LIN {X 0,Y 262.257,Z 673.457,A -85,B 0,C 180,E1 -18836.778,E2 -18836.778} C_VEL
LIN {X 0,Y 264.045,Z 616.117,A -85,B 0,C 180,E1 -18838.311,E2 -18838.311} C_VEL
LIN {X 0,Y 260.574,Z 590.625,A -85,B 0,C 180,E1 -18839.463,E2 -18839.463} C_VEL
LIN {X 0,Y 259.509,Z 585.684,A -85,B 0,C 180,E1 -18839.736,E2 -18839.736} C_VEL
LIN {X 0,Y 253.189,Z 570.092,A -85,B 0,C 180,E1 -18840.985,E2 -18840.985} C_VEL
LIN {X 0,Y 252.204,Z 567.395,A -85,B 0,C 180,E1 -18841.255,E2 -18841.255} C_VEL
LIN {X 0,Y 250.326,Z 558.805,A -85,B 0,C 180,E1 -18844.748,E2 -18844.748} C_VEL
LIN {X 0,Y 249.114,Z 553.456,A -85,B 0,C 180,E1 -18847.086,E2 -18847.086} C_VEL
LIN {X 0,Y 249.024,Z 553.465,A -85,B 0,C 180,E1 -18850.473,E2 -18850.473} C_VEL
LIN {X 0,Y 249.007,Z 553.466,A -85,B 0,C 180,E1 -18854.877,E2 -18854.877} C_VEL
LIN {X 0,Y 249.027,Z 553.464,A -85,B 0,C 180,E1 -18857.365,E2 -18857.365} C_VEL
LIN {X 0,Y 249.047,Z 553.463,A -85,B 0,C 180,E1 -18861.623,E2 -18861.623} C_VEL
LIN {X 0,Y 249.057,Z 553.461,A -85,B 0,C 180,E1 -18865.642,E2 -18865.642} C_VEL
LIN {X 0,Y 249.048,Z 553.464,A -85,B 0,C 180,E1 -18869.473,E2 -18869.473} C_VEL
LIN {X 0,Y 249.065,Z 553.457,A -85,B 0,C 180,E1 -18873.161,E2 -18873.161} C_VEL
LIN {X 0,Y 249.056,Z 553.455,A -85,B 0,C 180,E1 -18876.73,E2 -18876.73} C_VEL
LIN {X 0,Y 249.102,Z 553.454,A -85,B 0,C 180,E1 -18880.211,E2 -18880.211} C_VEL
LIN {X 0,Y 249.218,Z 553.438,A -85,B 0,C 180,E1 -18883.62,E2 -18883.62} C_VEL
LIN {X 0,Y 249.247,Z 553.429,A -85,B 0,C 180,E1 -18888.616,E2 -18888.616} C_VEL
LIN {X 0,Y 249.474,Z 553.409,A -85,B 0,C 180,E1 -18891.903,E2 -18891.903} C_VEL
LIN {X 0,Y 249.43,Z 553.409,A -85,B 0,C 180,E1 -18896.77,E2 -18896.77} C_VEL
LIN {X 0,Y 249.722,Z 553.376,A -85,B 0,C 180,E1 -18900,E2 -18900} C_VEL
LIN {X 0,Y 249.43,Z 553.406,A -85,B 0,C 180,E1 -18903.231,E2 -18903.231} C_VEL
LIN {X 0,Y 249.436,Z 553.41,A -85,B 0,C 180,E1 -18906.71,E2 -18906.71} C_VEL
LIN {X 0,Y 249.338,Z 553.412,A -85,B 0,C 180,E1 -18909.737,E2 -18909.737} C_VEL
LIN {X 0,Y 249.196,Z 553.442,A -85,B 0,C 180,E1 -18914.704,E2 -18914.704} C_VEL
LIN {X 0,Y 249.134,Z 553.444,A -85,B 0,C 180,E1 -18918.078,E2 -18918.078} C_VEL
LIN {X 0,Y 249.084,Z 553.449,A -85,B 0,C 180,E1 -18921.519,E2 -18921.519} C_VEL
LIN {X 0,Y 249.127,Z 553.451,A -85,B 0,C 180,E1 -18925.483,E2 -18925.483} C_VEL
LIN {X 0,Y 249.08,Z 553.458,A -85,B 0,C 180,E1 -18928.994,E2 -18928.994} C_VEL
LIN {X 0,Y 249.033,Z 553.461,A -85,B 0,C 180,E1 -18932.426,E2 -18932.426} C_VEL
LIN {X 0,Y 249.065,Z 553.451,A -85,B 0,C 180,E1 -18936.34,E2 -18936.34} C_VEL
LIN {X 0,Y 249.026,Z 553.463,A -85,B 0,C 180,E1 -18940.475,E2 -18940.475} C_VEL
LIN {X 0,Y 249.018,Z 553.466,A -85,B 0,C 180,E1 -18944.876,E2 -18944.876} C_VEL
LIN {X 0,Y 249.061,Z 553.462,A -85,B 0,C 180,E1 -18947.374,E2 -18947.374} C_VEL
LIN {X 0,Y 249.053,Z 553.46,A -85,B 0,C 180,E1 -18951.625,E2 -18951.625} C_VEL
LIN {X 0,Y 249.062,Z 553.46,A -85,B 0,C 180,E1 -18955.643,E2 -18955.643} C_VEL
LIN {X 0,Y 249.053,Z 553.464,A -85,B 0,C 180,E1 -18959.474,E2 -18959.474} C_VEL
LIN {X 0,Y 249.126,Z 553.516,A -85,B 0,C 180,E1 -18961.618,E2 -18961.618} C_VEL
LIN {X 0,Y 249.669,Z 555.641,A -85,B 0,C 180,E1 -18962.555,E2 -18962.555} C_VEL
LIN {X 0,Y 258.002,Z 574.299,A -85,B 0,C 180,E1 -18964.192,E2 -18964.192} C_VEL
LIN {X 0,Y 264.581,Z 591.655,A -85,B 0,C 180,E1 -18965.475,E2 -18965.475} C_VEL
LIN {X 0,Y 264.668,Z 597.246,A -85,B 0,C 180,E1 -18965.651,E2 -18965.651} C_VEL
LIN {X 0,Y 262.519,Z 662.1,A -85,B 0,C 180,E1 -18967.389,E2 -18967.389} C_VEL
LIN {X 0,Y 261.67,Z 674.994,A -85,B 0,C 180,E1 -18968.017,E2 -18968.017} C_VEL
LIN {X 0,Y 260.478,Z 687.741,A -85,B 0,C 180,E1 -18968.95,E2 -18968.95} C_VEL
LIN {X 0,Y 258.823,Z 699.889,A -85,B 0,C 180,E1 -18970.159,E2 -18970.159} C_VEL
LIN {X 0,Y 257.099,Z 711.369,A -85,B 0,C 180,E1 -18971.678,E2 -18971.678} C_VEL
LIN {X 0,Y 255.207,Z 721.715,A -85,B 0,C 180,E1 -18973.399,E2 -18973.399} C_VEL
LIN {X 0,Y 253.426,Z 730.182,A -85,B 0,C 180,E1 -18975.137,E2 -18975.137} C_VEL
LIN {X 0,Y 251.969,Z 737.973,A -85,B 0,C 180,E1 -18977.107,E2 -18977.107} C_VEL
LIN {X 0,Y 250.533,Z 745.289,A -85,B 0,C 180,E1 -18979.383,E2 -18979.383} C_VEL
LIN {X 0,Y 249.222,Z 751.71,A -85,B 0,C 180,E1 -18981.895,E2 -18981.895} C_VEL
LIN {X 0,Y 248.21,Z 756.578,A -85,B 0,C 180,E1 -18984.313,E2 -18984.313} C_VEL
LIN {X 0,Y 247.435,Z 760.339,A -85,B 0,C 180,E1 -18986.744,E2 -18986.744} C_VEL
LIN {X 0,Y 247.176,Z 762.276,A -85,B 0,C 180,E1 -18988.371,E2 -18988.371} C_VEL
LIN {X 0,Y 247.031,Z 763.804,A -85,B 0,C 180,E1 -18990,E2 -18990} C_VEL
LIN {X 0,Y 246.982,Z 764.891,A -85,B 0,C 180,E1 -18991.631,E2 -18991.631} C_VEL
LIN {X 0,Y 246.929,Z 765.58,A -85,B 0,C 180,E1 -18993.263,E2 -18993.263} C_VEL
LIN {X 0,Y 246.946,Z 765.908,A -85,B 0,C 180,E1 -18995.063,E2 -18995.063} C_VEL
LIN {X 0,Y 247.097,Z 765.335,A -85,B 0,C 180,E1 -18998.176,E2 -18998.176} C_VEL
LIN {X 0,Y 247.641,Z 763.152,A -85,B 0,C 180,E1 -19001.458,E2 -19001.458} C_VEL
LIN {X 0,Y 248.453,Z 760.413,A -85,B 0,C 180,E1 -19003.912,E2 -19003.912} C_VEL
LIN {X 0,Y 249.557,Z 756.648,A -85,B 0,C 180,E1 -19006.356,E2 -19006.356} C_VEL
LIN {X 0,Y 250.927,Z 751.748,A -85,B 0,C 180,E1 -19008.789,E2 -19008.789} C_VEL
LIN {X 0,Y 252.776,Z 745.563,A -85,B 0,C 180,E1 -19011.188,E2 -19011.188} C_VEL
LIN {X 0,Y 255.064,Z 737.823,A -85,B 0,C 180,E1 -19013.548,E2 -19013.548} C_VEL
LIN {X 0,Y 257.084,Z 729.651,A -85,B 0,C 180,E1 -19015.559,E2 -19015.559} C_VEL
LIN {X 0,Y 259.657,Z 719.105,A -85,B 0,C 180,E1 -19017.613,E2 -19017.613} C_VEL
LIN {X 0,Y 262.078,Z 707.972,A -85,B 0,C 180,E1 -19019.3,E2 -19019.3} C_VEL
LIN {X 0,Y 264.16,Z 697.037,A -85,B 0,C 180,E1 -19020.585,E2 -19020.585} C_VEL
LIN {X 0,Y 265.809,Z 684.913,A -85,B 0,C 180,E1 -19021.701,E2 -19021.701} C_VEL
LIN {X 0,Y 267.279,Z 672.232,A -85,B 0,C 180,E1 -19022.515,E2 -19022.515} C_VEL
LIN {X 0,Y 268.122,Z 659.678,A -85,B 0,C 180,E1 -19023.043,E2 -19023.043} C_VEL
LIN {X 0,Y 270.333,Z 598.373,A -85,B 0,C 180,E1 -19024.656,E2 -19024.656} C_VEL
LIN {X 0,Y 262.528,Z 580.576,A -85,B 0,C 180,E1 -19026.328,E2 -19026.328} C_VEL
LIN {X 0,Y 255.474,Z 566.537,A -85,B 0,C 180,E1 -19027.89,E2 -19027.89} C_VEL
LIN {X 0,Y 251.234,Z 559.018,A -85,B 0,C 180,E1 -19028.855,E2 -19028.855} C_VEL
LIN {X 0,Y 249.654,Z 555.862,A -85,B 0,C 180,E1 -19029.271,E2 -19029.271} C_VEL
LIN {X 0,Y 249.064,Z 553.462,A -85,B 0,C 180,E1 -19030.598,E2 -19030.598} C_VEL
LIN {X 0,Y 249.021,Z 553.465,A -85,B 0,C 180,E1 -19034.874,E2 -19034.874} C_VEL
LIN {X 0,Y 249.052,Z 553.456,A -85,B 0,C 180,E1 -19037.37,E2 -19037.37} C_VEL
LIN {X 0,Y 249.063,Z 553.46,A -85,B 0,C 180,E1 -19042.193,E2 -19042.193} C_VEL
LIN {X 0,Y 249.059,Z 553.457,A -85,B 0,C 180,E1 -19045.641,E2 -19045.641} C_VEL
LIN {X 0,Y 249.049,Z 553.454,A -85,B 0,C 180,E1 -19049.472,E2 -19049.472} C_VEL
LIN {X 0,Y 249.07,Z 553.451,A -85,B 0,C 180,E1 -19053.161,E2 -19053.161} C_VEL
LIN {X 0,Y 249.075,Z 553.453,A -85,B 0,C 180,E1 -19056.732,E2 -19056.732} C_VEL
LIN {X 0,Y 249.106,Z 553.456,A -85,B 0,C 180,E1 -19060.211,E2 -19060.211} C_VEL
LIN {X 0,Y 249.238,Z 553.436,A -85,B 0,C 180,E1 -19063.621,E2 -19063.621} C_VEL
LIN {X 0,Y 249.239,Z 553.433,A -85,B 0,C 180,E1 -19068.616,E2 -19068.616} C_VEL
LIN {X 0,Y 249.449,Z 553.402,A -85,B 0,C 180,E1 -19071.902,E2 -19071.902} C_VEL
LIN {X 0,Y 249.293,Z 553.432,A -85,B 0,C 180,E1 -19075.148,E2 -19075.148} C_VEL
LIN {X 0,Y 249.671,Z 553.373,A -85,B 0,C 180,E1 -19078.387,E2 -19078.387} C_VEL
LIN {X 0,Y 249.67,Z 553.382,A -85,B 0,C 180,E1 -19081.613,E2 -19081.613} C_VEL
LIN {X 0,Y 249.423,Z 553.408,A -85,B 0,C 180,E1 -19087.191,E2 -19087.191} C_VEL
LIN {X 0,Y 248.731,Z 553.493,A -85,B 0,C 180,E1 -19088.537,E2 -19088.537} C_VEL
LIN {X 0,Y 245.778,Z 553.87,A -85,B 0,C 180,E1 -19090.729,E2 -19090.729} C_VEL
LIN {X 0,Y 243.276,Z 554.174,A -85,B 0,C 180,E1 -19092.515,E2 -19092.515} C_VEL
LIN {X 0,Y 242.212,Z 554.302,A -85,B 0,C 180,E1 -19093.903,E2 -19093.903} C_VEL
LIN {X 0,Y 242.131,Z 554.314,A -85,B 0,C 180,E1 -19094.374,E2 -19094.374} C_VEL
LIN {X 0,Y 242.146,Z 554.32,A -85,B 0,C 180,E1 -19096.872,E2 -19096.872} C_VEL
LIN {X 0,Y 242.021,Z 554.336,A -85,B 0,C 180,E1 -19101.687,E2 -19101.687} C_VEL
LIN {X 0,Y 242.062,Z 554.332,A -85,B 0,C 180,E1 -19105.838,E2 -19105.838} C_VEL
LIN {X 0,Y 242.026,Z 554.336,A -85,B 0,C 180,E1 -19109.581,E2 -19109.581} C_VEL
LIN {X 0,Y 241.987,Z 554.341,A -85,B 0,C 180,E1 -19113.491,E2 -19113.491} C_VEL
LIN {X 0,Y 242.008,Z 554.339,A -85,B 0,C 180,E1 -19117.578,E2 -19117.578} C_VEL
LIN {X 0,Y 241.953,Z 554.348,A -85,B 0,C 180,E1 -19121.919,E2 -19121.919} C_VEL
LIN {X 0,Y 241.935,Z 554.351,A -85,B 0,C 180,E1 -19126.571,E2 -19126.571} C_VEL
LIN {X 0,Y 241.991,Z 554.486,A -85,B 0,C 180,E1 -19127.942,E2 -19127.942} C_VEL
LIN {X 0,Y 244.207,Z 562.602,A -85,B 0,C 180,E1 -19132.006,E2 -19132.006} C_VEL
LIN {X 0,Y 245.342,Z 567.185,A -85,B 0,C 180,E1 -19134.048,E2 -19134.048} C_VEL
LIN {X 0,Y 254.461,Z 585.606,A -85,B 0,C 180,E1 -19136.239,E2 -19136.239} C_VEL
LIN {X 0,Y 260.641,Z 599.85,A -85,B 0,C 180,E1 -19137.663,E2 -19137.663} C_VEL
LIN {X 0,Y 263.653,Z 619.289,A -85,B 0,C 180,E1 -19138.723,E2 -19138.723} C_VEL
LIN {X 0,Y 261.5,Z 675.447,A -85,B 0,C 180,E1 -19140.247,E2 -19140.247} C_VEL
LIN {X 0,Y 260.259,Z 688.736,A -85,B 0,C 180,E1 -19140.872,E2 -19140.872} C_VEL
LIN {X 0,Y 258.437,Z 701.888,A -85,B 0,C 180,E1 -19141.804,E2 -19141.804} C_VEL
LIN {X 0,Y 256.5,Z 713.038,A -85,B 0,C 180,E1 -19142.902,E2 -19142.902} C_VEL
LIN {X 0,Y 254.106,Z 724.62,A -85,B 0,C 180,E1 -19144.396,E2 -19144.396} C_VEL
LIN {X 0,Y 251.548,Z 735.052,A -85,B 0,C 180,E1 -19146.102,E2 -19146.102} C_VEL
LIN {X 0,Y 249.025,Z 744.458,A -85,B 0,C 180,E1 -19148.042,E2 -19148.042} C_VEL
LIN {X 0,Y 246.902,Z 752.18,A -85,B 0,C 180,E1 -19150.028,E2 -19150.028} C_VEL
LIN {X 0,Y 244.783,Z 759.746,A -85,B 0,C 180,E1 -19152.455,E2 -19152.455} C_VEL
LIN {X 0,Y 242.964,Z 765.844,A -85,B 0,C 180,E1 -19154.91,E2 -19154.91} C_VEL
LIN {X 0,Y 241.589,Z 770.69,A -85,B 0,C 180,E1 -19157.398,E2 -19157.398} C_VEL
LIN {X 0,Y 240.678,Z 774.427,A -85,B 0,C 180,E1 -19159.91,E2 -19159.91} C_VEL
LIN {X 0,Y 240.233,Z 776.363,A -85,B 0,C 180,E1 -19161.589,E2 -19161.589} C_VEL
LIN {X 0,Y 239.956,Z 777.877,A -85,B 0,C 180,E1 -19163.272,E2 -19163.272} C_VEL
LIN {X 0,Y 239.769,Z 779.626,A -85,B 0,C 180,E1 -19166.639,E2 -19166.639} C_VEL
LIN {X 0,Y 239.837,Z 779.923,A -85,B 0,C 180,E1 -19168.321,E2 -19168.321} C_VEL
LIN {X 0,Y 239.915,Z 779.827,A -85,B 0,C 180,E1 -19170,E2 -19170} C_VEL
LIN {X 0,Y 239.841,Z 779.29,A -85,B 0,C 180,E1 -19171.679,E2 -19171.679} C_VEL
LIN {X 0,Y 239.84,Z 777.123,A -85,B 0,C 180,E1 -19174.931,E2 -19174.931} C_VEL
LIN {X 0,Y 240.045,Z 774.202,A -85,B 0,C 180,E1 -19177.571,E2 -19177.571} C_VEL
LIN {X 0,Y 240.553,Z 770.345,A -85,B 0,C 180,E1 -19180.096,E2 -19180.096} C_VEL
LIN {X 0,Y 241.388,Z 765.354,A -85,B 0,C 180,E1 -19182.613,E2 -19182.613} C_VEL
LIN {X 0,Y 242.695,Z 759.08,A -85,B 0,C 180,E1 -19185.107,E2 -19185.107} C_VEL
LIN {X 0,Y 244.409,Z 751.231,A -85,B 0,C 180,E1 -19187.573,E2 -19187.573} C_VEL
LIN {X 0,Y 246.082,Z 742.93,A -85,B 0,C 180,E1 -19189.674,E2 -19189.674} C_VEL
LIN {X 0,Y 247.92,Z 733.413,A -85,B 0,C 180,E1 -19191.624,E2 -19191.624} C_VEL
LIN {X 0,Y 249.979,Z 722.522,A -85,B 0,C 180,E1 -19193.397,E2 -19193.397} C_VEL
LIN {X 0,Y 251.772,Z 711.865,A -85,B 0,C 180,E1 -19194.753,E2 -19194.753} C_VEL
LIN {X 0,Y 253.45,Z 700.16,A -85,B 0,C 180,E1 -19195.895,E2 -19195.895} C_VEL
LIN {X 0,Y 254.928,Z 686.874,A -85,B 0,C 180,E1 -19196.835,E2 -19196.835} C_VEL
LIN {X 0,Y 255.794,Z 674.748,A -85,B 0,C 180,E1 -19197.4,E2 -19197.4} C_VEL
LIN {X 0,Y 257.705,Z 617.043,A -85,B 0,C 180,E1 -19198.982,E2 -19198.982} C_VEL
LIN {X 0,Y 253.937,Z 589.557,A -85,B 0,C 180,E1 -19200.278,E2 -19200.278} C_VEL
LIN {X 0,Y 247.922,Z 574.236,A -85,B 0,C 180,E1 -19201.526,E2 -19201.526} C_VEL
LIN {X 0,Y 244.945,Z 567.249,A -85,B 0,C 180,E1 -19202.186,E2 -19202.186} C_VEL
LIN {X 0,Y 243.05,Z 558.388,A -85,B 0,C 180,E1 -19205.939,E2 -19205.939} C_VEL
LIN {X 0,Y 242.015,Z 554.34,A -85,B 0,C 180,E1 -19207.772,E2 -19207.772} C_VEL
LIN {X 0,Y 241.942,Z 554.346,A -85,B 0,C 180,E1 -19211.92,E2 -19211.92} C_VEL
LIN {X 0,Y 241.942,Z 554.344,A -85,B 0,C 180,E1 -19216.568,E2 -19216.568} C_VEL
LIN {X 0,Y 241.985,Z 554.34,A -85,B 0,C 180,E1 -19220.287,E2 -19220.287} C_VEL
LIN {X 0,Y 242.033,Z 554.334,A -85,B 0,C 180,E1 -19224.497,E2 -19224.497} C_VEL
LIN {X 0,Y 241.972,Z 554.341,A -85,B 0,C 180,E1 -19228.48,E2 -19228.48} C_VEL
LIN {X 0,Y 242.002,Z 554.334,A -85,B 0,C 180,E1 -19232.312,E2 -19232.312} C_VEL
LIN {X 0,Y 242.036,Z 554.33,A -85,B 0,C 180,E1 -19236.014,E2 -19236.014} C_VEL
LIN {X 0,Y 242.03,Z 554.338,A -85,B 0,C 180,E1 -19239.607,E2 -19239.607} C_VEL
LIN {X 0,Y 242.159,Z 554.314,A -85,B 0,C 180,E1 -19243.278,E2 -19243.278} C_VEL
LIN {X 0,Y 242.18,Z 554.309,A -85,B 0,C 180,E1 -19248.28,E2 -19248.28} C_VEL
LIN {X 0,Y 242.421,Z 554.289,A -85,B 0,C 180,E1 -19251.666,E2 -19251.666} C_VEL
LIN {X 0,Y 242.253,Z 554.301,A -85,B 0,C 180,E1 -19255.007,E2 -19255.007} C_VEL
LIN {X 0,Y 242.631,Z 554.26,A -85,B 0,C 180,E1 -19258.34,E2 -19258.34} C_VEL
LIN {X 0,Y 242.631,Z 554.253,A -85,B 0,C 180,E1 -19261.66,E2 -19261.66} C_VEL
LIN {X 0,Y 242.417,Z 554.287,A -85,B 0,C 180,E1 -19266.682,E2 -19266.682} C_VEL
LIN {X 0,Y 242.262,Z 554.291,A -85,B 0,C 180,E1 -19270.024,E2 -19270.024} C_VEL
LIN {X 0,Y 242.159,Z 554.32,A -85,B 0,C 180,E1 -19275.142,E2 -19275.142} C_VEL
LIN {X 0,Y 242.068,Z 554.323,A -85,B 0,C 180,E1 -19278.625,E2 -19278.625} C_VEL
LIN {X 0,Y 242.01,Z 554.335,A -85,B 0,C 180,E1 -19282.181,E2 -19282.181} C_VEL
LIN {X 0,Y 242.063,Z 554.328,A -85,B 0,C 180,E1 -19285.839,E2 -19285.839} C_VEL
LIN {X 0,Y 242.027,Z 554.337,A -85,B 0,C 180,E1 -19289.581,E2 -19289.581} C_VEL
LIN {X 0,Y 241.988,Z 554.344,A -85,B 0,C 180,E1 -19293.492,E2 -19293.492} C_VEL
LIN {X 0,Y 241.996,Z 554.325,A -85,B 0,C 180,E1 -19297.581,E2 -19297.581} C_VEL
LIN {X 0,Y 241.951,Z 554.345,A -85,B 0,C 180,E1 -19301.92,E2 -19301.92} C_VEL
LIN {X 0,Y 241.99,Z 554.338,A -85,B 0,C 180,E1 -19306.558,E2 -19306.558} C_VEL
LIN {X 0,Y 242.008,Z 554.337,A -85,B 0,C 180,E1 -19310.292,E2 -19310.292} C_VEL
LIN {X 0,Y 242.037,Z 554.335,A -85,B 0,C 180,E1 -19314.499,E2 -19314.499} C_VEL
LIN {X 0,Y 241.977,Z 554.345,A -85,B 0,C 180,E1 -19318.481,E2 -19318.481} C_VEL
LIN {X 0,Y 242.044,Z 554.361,A -85,B 0,C 180,E1 -19320.899,E2 -19320.899} C_VEL
LIN {X 0,Y 242.432,Z 555.851,A -85,B 0,C 180,E1 -19321.575,E2 -19321.575} C_VEL
LIN {X 0,Y 250.422,Z 573.112,A -85,B 0,C 180,E1 -19323.218,E2 -19323.218} C_VEL
LIN {X 0,Y 258.393,Z 593.558,A -85,B 0,C 180,E1 -19324.833,E2 -19324.833} C_VEL
LIN {X 0,Y 256.709,Z 646.367,A -85,B 0,C 180,E1 -19326.261,E2 -19326.261} C_VEL
LIN {X 0,Y 255.975,Z 664.604,A -85,B 0,C 180,E1 -19326.818,E2 -19326.818} C_VEL
LIN {X 0,Y 255.025,Z 677.674,A -85,B 0,C 180,E1 -19327.52,E2 -19327.52} C_VEL
LIN {X 0,Y 253.741,Z 689.696,A -85,B 0,C 180,E1 -19328.47,E2 -19328.47} C_VEL
LIN {X 0,Y 252.186,Z 700.594,A -85,B 0,C 180,E1 -19329.614,E2 -19329.614} C_VEL
LIN {X 0,Y 250.409,Z 711.981,A -85,B 0,C 180,E1 -19331.171,E2 -19331.171} C_VEL
LIN {X 0,Y 248.444,Z 722.258,A -85,B 0,C 180,E1 -19332.933,E2 -19332.933} C_VEL
LIN {X 0,Y 246.599,Z 730.667,A -85,B 0,C 180,E1 -19334.715,E2 -19334.715} C_VEL
LIN {X 0,Y 244.786,Z 739.759,A -85,B 0,C 180,E1 -19337.144,E2 -19337.144} C_VEL
LIN {X 0,Y 243.447,Z 746.28,A -85,B 0,C 180,E1 -19339.303,E2 -19339.303} C_VEL
LIN {X 0,Y 242.21,Z 752.058,A -85,B 0,C 180,E1 -19341.658,E2 -19341.658} C_VEL
LIN {X 0,Y 241.174,Z 756.894,A -85,B 0,C 180,E1 -19344.146,E2 -19344.146} C_VEL
LIN {X 0,Y 240.377,Z 760.627,A -85,B 0,C 180,E1 -19346.648,E2 -19346.648} C_VEL
LIN {X 0,Y 240.107,Z 762.551,A -85,B 0,C 180,E1 -19348.323,E2 -19348.323} C_VEL
LIN {X 0,Y 239.96,Z 764.062,A -85,B 0,C 180,E1 -19350,E2 -19350} C_VEL
LIN {X 0,Y 239.89,Z 765.127,A -85,B 0,C 180,E1 -19351.679,E2 -19351.679} C_VEL
LIN {X 0,Y 239.842,Z 766.091,A -85,B 0,C 180,E1 -19354.931,E2 -19354.931} C_VEL
LIN {X 0,Y 239.882,Z 766.02,A -85,B 0,C 180,E1 -19356.73,E2 -19356.73} C_VEL
LIN {X 0,Y 240.028,Z 765.508,A -85,B 0,C 180,E1 -19358.418,E2 -19358.418} C_VEL
LIN {X 0,Y 240.279,Z 764.6,A -85,B 0,C 180,E1 -19360.107,E2 -19360.107} C_VEL
LIN {X 0,Y 240.625,Z 763.3,A -85,B 0,C 180,E1 -19361.797,E2 -19361.797} C_VEL
LIN {X 0,Y 241.502,Z 760.534,A -85,B 0,C 180,E1 -19364.321,E2 -19364.321} C_VEL
LIN {X 0,Y 242.932,Z 755.913,A -85,B 0,C 180,E1 -19367.313,E2 -19367.313} C_VEL
LIN {X 0,Y 244.767,Z 749.88,A -85,B 0,C 180,E1 -19370.154,E2 -19370.154} C_VEL
LIN {X 0,Y 246.806,Z 743.163,A -85,B 0,C 180,E1 -19372.607,E2 -19372.607} C_VEL
LIN {X 0,Y 249.313,Z 734.801,A -85,B 0,C 180,E1 -19375.013,E2 -19375.013} C_VEL
LIN {X 0,Y 251.562,Z 726.156,A -85,B 0,C 180,E1 -19376.999,E2 -19376.999} C_VEL
LIN {X 0,Y 253.909,Z 716.664,A -85,B 0,C 180,E1 -19378.745,E2 -19378.745} C_VEL
LIN {X 0,Y 256.153,Z 706.289,A -85,B 0,C 180,E1 -19380.274,E2 -19380.274} C_VEL
LIN {X 0,Y 258.34,Z 694.903,A -85,B 0,C 180,E1 -19381.579,E2 -19381.579} C_VEL
LIN {X 0,Y 259.93,Z 683.165,A -85,B 0,C 180,E1 -19382.62,E2 -19382.62} C_VEL
LIN {X 0,Y 261.365,Z 669.999,A -85,B 0,C 180,E1 -19383.425,E2 -19383.425} C_VEL
LIN {X 0,Y 262.209,Z 657.215,A -85,B 0,C 180,E1 -19383.916,E2 -19383.916} C_VEL
LIN {X 0,Y 264.345,Z 600.475,A -85,B 0,C 180,E1 -19385.423,E2 -19385.423} C_VEL
LIN {X 0,Y 257.486,Z 584.678,A -85,B 0,C 180,E1 -19386.96,E2 -19386.96} C_VEL
LIN {X 0,Y 250.232,Z 570.136,A -85,B 0,C 180,E1 -19388.637,E2 -19388.637} C_VEL
LIN {X 0,Y 243.958,Z 559.102,A -85,B 0,C 180,E1 -19390.144,E2 -19390.144} C_VEL
LIN {X 0,Y 242.451,Z 556.033,A -85,B 0,C 180,E1 -19390.61,E2 -19390.61} C_VEL
LIN {X 0,Y 242.059,Z 554.332,A -85,B 0,C 180,E1 -19391.629,E2 -19391.629} C_VEL
LIN {X 0,Y 241.985,Z 554.344,A -85,B 0,C 180,E1 -19396.557,E2 -19396.557} C_VEL
LIN {X 0,Y 241.98,Z 554.332,A -85,B 0,C 180,E1 -19400.285,E2 -19400.285} C_VEL
LIN {X 0,Y 242.034,Z 554.337,A -85,B 0,C 180,E1 -19404.497,E2 -19404.497} C_VEL
LIN {X 0,Y 241.973,Z 554.342,A -85,B 0,C 180,E1 -19408.479,E2 -19408.479} C_VEL
LIN {X 0,Y 242.005,Z 554.337,A -85,B 0,C 180,E1 -19412.312,E2 -19412.312} C_VEL
LIN {X 0,Y 242.053,Z 554.334,A -85,B 0,C 180,E1 -19416.015,E2 -19416.015} C_VEL
LIN {X 0,Y 242.033,Z 554.336,A -85,B 0,C 180,E1 -19419.607,E2 -19419.607} C_VEL
LIN {X 0,Y 242.159,Z 554.314,A -85,B 0,C 180,E1 -19423.278,E2 -19423.278} C_VEL
LIN {X 0,Y 242.176,Z 554.31,A -85,B 0,C 180,E1 -19428.279,E2 -19428.279} C_VEL
LIN {X 0,Y 242.395,Z 554.282,A -85,B 0,C 180,E1 -19431.664,E2 -19431.664} C_VEL
LIN {X 0,Y 242.253,Z 554.31,A -85,B 0,C 180,E1 -19435.007,E2 -19435.007} C_VEL
LIN {X 0,Y 242.631,Z 554.249,A -85,B 0,C 180,E1 -19438.34,E2 -19438.34} C_VEL
LIN {X 0,Y 242.631,Z 554.259,A -85,B 0,C 180,E1 -19441.66,E2 -19441.66} C_VEL
LIN {X 0,Y 242.389,Z 554.284,A -85,B 0,C 180,E1 -19447.177,E2 -19447.177} C_VEL
LIN {X 0,Y 242.262,Z 554.303,A -85,B 0,C 180,E1 -19450.024,E2 -19450.024} C_VEL
LIN {X 0,Y 242.131,Z 554.314,A -85,B 0,C 180,E1 -19454.374,E2 -19454.374} C_VEL
LIN {X 0,Y 241.465,Z 554.408,A -85,B 0,C 180,E1 -19455.763,E2 -19455.763} C_VEL
LIN {X 0,Y 238.573,Z 554.77,A -85,B 0,C 180,E1 -19458.026,E2 -19458.026} C_VEL
LIN {X 0,Y 236.109,Z 555.075,A -85,B 0,C 180,E1 -19459.87,E2 -19459.87} C_VEL
LIN {X 0,Y 235.055,Z 555.204,A -85,B 0,C 180,E1 -19461.302,E2 -19461.302} C_VEL
LIN {X 0,Y 234.971,Z 555.211,A -85,B 0,C 180,E1 -19461.788,E2 -19461.788} C_VEL
LIN {X 0,Y 234.99,Z 555.208,A -85,B 0,C 180,E1 -19466.207,E2 -19466.207} C_VEL
LIN {X 0,Y 234.928,Z 555.22,A -85,B 0,C 180,E1 -19470.568,E2 -19470.568} C_VEL
LIN {X 0,Y 234.957,Z 555.217,A -85,B 0,C 180,E1 -19474.633,E2 -19474.633} C_VEL
LIN {X 0,Y 234.964,Z 555.218,A -85,B 0,C 180,E1 -19478.953,E2 -19478.953} C_VEL
LIN {X 0,Y 234.92,Z 555.225,A -85,B 0,C 180,E1 -19483.478,E2 -19483.478} C_VEL
LIN {X 0,Y 234.898,Z 555.244,A -85,B 0,C 180,E1 -19486.751,E2 -19486.751} C_VEL
LIN {X 0,Y 237.424,Z 564.45,A -85,B 0,C 180,E1 -19491.566,E2 -19491.566} C_VEL
LIN {X 0,Y 238.047,Z 566.88,A -85,B 0,C 180,E1 -19492.671,E2 -19492.671} C_VEL
LIN {X 0,Y 240.252,Z 571.044,A -85,B 0,C 180,E1 -19493.251,E2 -19493.251} C_VEL
LIN {X 0,Y 248.781,Z 588.132,A -85,B 0,C 180,E1 -19495.393,E2 -19495.393} C_VEL
LIN {X 0,Y 254.987,Z 602.592,A -85,B 0,C 180,E1 -19496.895,E2 -19496.895} C_VEL
LIN {X 0,Y 257.711,Z 620.887,A -85,B 0,C 180,E1 -19497.917,E2 -19497.917} C_VEL
LIN {X 0,Y 255.469,Z 675.326,A -85,B 0,C 180,E1 -19499.416,E2 -19499.416} C_VEL
LIN {X 0,Y 254.187,Z 688.671,A -85,B 0,C 180,E1 -19500.059,E2 -19500.059} C_VEL
LIN {X 0,Y 252.391,Z 701.138,A -85,B 0,C 180,E1 -19500.952,E2 -19500.952} C_VEL
LIN {X 0,Y 250.204,Z 713.237,A -85,B 0,C 180,E1 -19502.162,E2 -19502.162} C_VEL
LIN {X 0,Y 247.726,Z 724.744,A -85,B 0,C 180,E1 -19503.687,E2 -19503.687} C_VEL
LIN {X 0,Y 245.081,Z 735.119,A -85,B 0,C 180,E1 -19505.431,E2 -19505.431} C_VEL
LIN {X 0,Y 242.445,Z 744.462,A -85,B 0,C 180,E1 -19507.413,E2 -19507.413} C_VEL
LIN {X 0,Y 239.894,Z 753.39,A -85,B 0,C 180,E1 -19509.829,E2 -19509.829} C_VEL
LIN {X 0,Y 237.702,Z 760.8,A -85,B 0,C 180,E1 -19512.359,E2 -19512.359} C_VEL
LIN {X 0,Y 235.528,Z 767.499,A -85,B 0,C 180,E1 -19515.308,E2 -19515.308} C_VEL
LIN {X 0,Y 234.281,Z 771.939,A -85,B 0,C 180,E1 -19517.879,E2 -19517.879} C_VEL
LIN {X 0,Y 233.675,Z 774.289,A -85,B 0,C 180,E1 -19519.604,E2 -19519.604} C_VEL
LIN {X 0,Y 233.201,Z 776.214,A -85,B 0,C 180,E1 -19521.334,E2 -19521.334} C_VEL
LIN {X 0,Y 232.893,Z 777.709,A -85,B 0,C 180,E1 -19523.067,E2 -19523.067} C_VEL
LIN {X 0,Y 232.677,Z 779.437,A -85,B 0,C 180,E1 -19526.537,E2 -19526.537} C_VEL
LIN {X 0,Y 232.749,Z 779.724,A -85,B 0,C 180,E1 -19528.27,E2 -19528.27} C_VEL
LIN {X 0,Y 232.824,Z 779.611,A -85,B 0,C 180,E1 -19530,E2 -19530} C_VEL
LIN {X 0,Y 232.753,Z 779.061,A -85,B 0,C 180,E1 -19531.73,E2 -19531.73} C_VEL
LIN {X 0,Y 232.753,Z 777.079,A -85,B 0,C 180,E1 -19534.837,E2 -19534.837} C_VEL
LIN {X 0,Y 233,Z 773.93,A -85,B 0,C 180,E1 -19537.801,E2 -19537.801} C_VEL
LIN {X 0,Y 233.535,Z 770.05,A -85,B 0,C 180,E1 -19540.402,E2 -19540.402} C_VEL
LIN {X 0,Y 234.41,Z 765.033,A -85,B 0,C 180,E1 -19542.994,E2 -19542.994} C_VEL
LIN {X 0,Y 235.827,Z 758.733,A -85,B 0,C 180,E1 -19545.558,E2 -19545.558} C_VEL
LIN {X 0,Y 237.638,Z 750.839,A -85,B 0,C 180,E1 -19548.091,E2 -19548.091} C_VEL
LIN {X 0,Y 239.27,Z 742.962,A -85,B 0,C 180,E1 -19550.143,E2 -19550.143} C_VEL
LIN {X 0,Y 241.302,Z 732.937,A -85,B 0,C 180,E1 -19552.248,E2 -19552.248} C_VEL
LIN {X 0,Y 243.474,Z 721.971,A -85,B 0,C 180,E1 -19554.061,E2 -19554.061} C_VEL
LIN {X 0,Y 245.314,Z 711.211,A -85,B 0,C 180,E1 -19555.45,E2 -19555.45} C_VEL
LIN {X 0,Y 247.077,Z 699.383,A -85,B 0,C 180,E1 -19556.615,E2 -19556.615} C_VEL
LIN {X 0,Y 248.508,Z 686.658,A -85,B 0,C 180,E1 -19557.529,E2 -19557.529} C_VEL
LIN {X 0,Y 249.399,Z 674.519,A -85,B 0,C 180,E1 -19558.107,E2 -19558.107} C_VEL
LIN {X 0,Y 251.342,Z 617.531,A -85,B 0,C 180,E1 -19559.708,E2 -19559.708} C_VEL
LIN {X 0,Y 247.844,Z 591.602,A -85,B 0,C 180,E1 -19560.971,E2 -19560.971} C_VEL
LIN {X 0,Y 241.706,Z 576.246,A -85,B 0,C 180,E1 -19562.295,E2 -19562.295} C_VEL
LIN {X 0,Y 237.713,Z 567.073,A -85,B 0,C 180,E1 -19563.187,E2 -19563.187} C_VEL
LIN {X 0,Y 235.761,Z 558.19,A -85,B 0,C 180,E1 -19567.131,E2 -19567.131} C_VEL
LIN {X 0,Y 234.942,Z 555.22,A -85,B 0,C 180,E1 -19568.641,E2 -19568.641} C_VEL
LIN {X 0,Y 234.888,Z 555.224,A -85,B 0,C 180,E1 -19573.484,E2 -19573.484} C_VEL
LIN {X 0,Y 234.92,Z 555.219,A -85,B 0,C 180,E1 -19576.522,E2 -19576.522} C_VEL
LIN {X 0,Y 234.952,Z 555.218,A -85,B 0,C 180,E1 -19581.085,E2 -19581.085} C_VEL
LIN {X 0,Y 234.957,Z 555.219,A -85,B 0,C 180,E1 -19585.367,E2 -19585.367} C_VEL
LIN {X 0,Y 234.965,Z 555.214,A -85,B 0,C 180,E1 -19590.157,E2 -19590.157} C_VEL
LIN {X 0,Y 234.99,Z 555.214,A -85,B 0,C 180,E1 -19593.793,E2 -19593.793} C_VEL
LIN {X 0,Y 234.993,Z 555.212,A -85,B 0,C 180,E1 -19598.968,E2 -19598.968} C_VEL
LIN {X 0,Y 235.091,Z 555.193,A -85,B 0,C 180,E1 -19603.06,E2 -19603.06} C_VEL
LIN {X 0,Y 235.112,Z 555.19,A -85,B 0,C 180,E1 -19607.922,E2 -19607.922} C_VEL
LIN {X 0,Y 235.371,Z 555.167,A -85,B 0,C 180,E1 -19611.414,E2 -19611.414} C_VEL
LIN {X 0,Y 235.397,Z 555.163,A -85,B 0,C 180,E1 -19613.141,E2 -19613.141} C_VEL
LIN {X 0,Y 235.59,Z 555.137,A -85,B 0,C 180,E1 -19618.291,E2 -19618.291} C_VEL
LIN {X 0,Y 235.59,Z 555.129,A -85,B 0,C 180,E1 -19621.71,E2 -19621.71} C_VEL
LIN {X 0,Y 235.388,Z 555.163,A -85,B 0,C 180,E1 -19626.859,E2 -19626.859} C_VEL
LIN {X 0,Y 235.209,Z 555.168,A -85,B 0,C 180,E1 -19630.328,E2 -19630.328} C_VEL
LIN {X 0,Y 235.107,Z 555.2,A -85,B 0,C 180,E1 -19635.607,E2 -19635.607} C_VEL
LIN {X 0,Y 235.004,Z 555.197,A -85,B 0,C 180,E1 -19639.206,E2 -19639.206} C_VEL
LIN {X 0,Y 234.958,Z 555.214,A -85,B 0,C 180,E1 -19642.883,E2 -19642.883} C_VEL
LIN {X 0,Y 234.967,Z 555.21,A -85,B 0,C 180,E1 -19646.658,E2 -19646.658} C_VEL
LIN {X 0,Y 234.929,Z 555.218,A -85,B 0,C 180,E1 -19650.568,E2 -19650.568} C_VEL
LIN {X 0,Y 234.958,Z 555.216,A -85,B 0,C 180,E1 -19654.634,E2 -19654.634} C_VEL
LIN {X 0,Y 234.94,Z 555.208,A -85,B 0,C 180,E1 -19658.945,E2 -19658.945} C_VEL
LIN {X 0,Y 234.924,Z 555.221,A -85,B 0,C 180,E1 -19663.478,E2 -19663.478} C_VEL
LIN {X 0,Y 234.964,Z 555.213,A -85,B 0,C 180,E1 -19666.533,E2 -19666.533} C_VEL
LIN {X 0,Y 234.955,Z 555.216,A -85,B 0,C 180,E1 -19671.087,E2 -19671.087} C_VEL
LIN {X 0,Y 234.961,Z 555.218,A -85,B 0,C 180,E1 -19675.368,E2 -19675.368} C_VEL
LIN {X 0,Y 234.99,Z 555.25,A -85,B 0,C 180,E1 -19680.15,E2 -19680.15} C_VEL
LIN {X 0,Y 235.138,Z 555.935,A -85,B 0,C 180,E1 -19680.488,E2 -19680.488} C_VEL
LIN {X 0,Y 236.872,Z 559.537,A -85,B 0,C 180,E1 -19680.896,E2 -19680.896} C_VEL
LIN {X 0,Y 243.411,Z 573.323,A -85,B 0,C 180,E1 -19682.298,E2 -19682.298} C_VEL
LIN {X 0,Y 250.811,Z 591.703,A -85,B 0,C 180,E1 -19683.864,E2 -19683.864} C_VEL
LIN {X 0,Y 252.121,Z 595.877,A -85,B 0,C 180,E1 -19684.158,E2 -19684.158} C_VEL
LIN {X 0,Y 249.689,Z 663.008,A -85,B 0,C 180,E1 -19686.041,E2 -19686.041} C_VEL
LIN {X 0,Y 248.729,Z 676.564,A -85,B 0,C 180,E1 -19686.754,E2 -19686.754} C_VEL
LIN {X 0,Y 247.321,Z 689.535,A -85,B 0,C 180,E1 -19687.772,E2 -19687.772} C_VEL
LIN {X 0,Y 245.574,Z 701.298,A -85,B 0,C 180,E1 -19689.039,E2 -19689.039} C_VEL
LIN {X 0,Y 243.743,Z 712.592,A -85,B 0,C 180,E1 -19690.635,E2 -19690.635} C_VEL
LIN {X 0,Y 241.702,Z 722.792,A -85,B 0,C 180,E1 -19692.442,E2 -19692.442} C_VEL
LIN {X 0,Y 239.377,Z 732.771,A -85,B 0,C 180,E1 -19694.679,E2 -19694.679} C_VEL
LIN {X 0,Y 237.633,Z 741.519,A -85,B 0,C 180,E1 -19697.185,E2 -19697.185} C_VEL
LIN {X 0,Y 236.026,Z 748.548,A -85,B 0,C 180,E1 -19699.709,E2 -19699.709} C_VEL
LIN {X 0,Y 234.838,Z 754.152,A -85,B 0,C 180,E1 -19702.261,E2 -19702.261} C_VEL
LIN {X 0,Y 233.79,Z 758.578,A -85,B 0,C 180,E1 -19704.826,E2 -19704.826} C_VEL
LIN {X 0,Y 233.321,Z 760.915,A -85,B 0,C 180,E1 -19706.546,E2 -19706.546} C_VEL
LIN {X 0,Y 233.04,Z 762.825,A -85,B 0,C 180,E1 -19708.272,E2 -19708.272} C_VEL
LIN {X 0,Y 232.889,Z 764.316,A -85,B 0,C 180,E1 -19710,E2 -19710} C_VEL
LIN {X 0,Y 232.8,Z 765.363,A -85,B 0,C 180,E1 -19711.73,E2 -19711.73} C_VEL
LIN {X 0,Y 232.736,Z 766.274,A -85,B 0,C 180,E1 -19714.783,E2 -19714.783} C_VEL
LIN {X 0,Y 232.798,Z 766.214,A -85,B 0,C 180,E1 -19716.936,E2 -19716.936} C_VEL
LIN {X 0,Y 233.244,Z 764.761,A -85,B 0,C 180,E1 -19720.415,E2 -19720.415} C_VEL
LIN {X 0,Y 233.62,Z 763.448,A -85,B 0,C 180,E1 -19722.156,E2 -19722.156} C_VEL
LIN {X 0,Y 234.565,Z 760.655,A -85,B 0,C 180,E1 -19724.754,E2 -19724.754} C_VEL
LIN {X 0,Y 235.991,Z 756.337,A -85,B 0,C 180,E1 -19727.637,E2 -19727.637} C_VEL
LIN {X 0,Y 237.406,Z 751.871,A -85,B 0,C 180,E1 -19729.903,E2 -19729.903} C_VEL
LIN {X 0,Y 239.456,Z 745.617,A -85,B 0,C 180,E1 -19732.429,E2 -19732.429} C_VEL
LIN {X 0,Y 242.013,Z 737.76,A -85,B 0,C 180,E1 -19734.902,E2 -19734.902} C_VEL
LIN {X 0,Y 244.26,Z 729.428,A -85,B 0,C 180,E1 -19737.024,E2 -19737.024} C_VEL
LIN {X 0,Y 246.8,Z 719.908,A -85,B 0,C 180,E1 -19738.953,E2 -19738.953} C_VEL
LIN {X 0,Y 249.419,Z 708.908,A -85,B 0,C 180,E1 -19740.711,E2 -19740.711} C_VEL
LIN {X 0,Y 251.623,Z 698.097,A -85,B 0,C 180,E1 -19742.051,E2 -19742.051} C_VEL
LIN {X 0,Y 253.446,Z 686.16,A -85,B 0,C 180,E1 -19743.206,E2 -19743.206} C_VEL
LIN {X 0,Y 255.115,Z 673.17,A -85,B 0,C 180,E1 -19744.088,E2 -19744.088} C_VEL
LIN {X 0,Y 256.029,Z 660.608,A -85,B 0,C 180,E1 -19744.65,E2 -19744.65} C_VEL
LIN {X 0,Y 258.359,Z 602.518,A -85,B 0,C 180,E1 -19746.236,E2 -19746.236} C_VEL
LIN {X 0,Y 252.327,Z 588.477,A -85,B 0,C 180,E1 -19747.652,E2 -19747.652} C_VEL
LIN {X 0,Y 245.349,Z 574.324,A -85,B 0,C 180,E1 -19749.338,E2 -19749.338} C_VEL
LIN {X 0,Y 239.092,Z 563.243,A -85,B 0,C 180,E1 -19750.909,E2 -19750.909} C_VEL
LIN {X 0,Y 236.896,Z 559.568,A -85,B 0,C 180,E1 -19751.48,E2 -19751.48} C_VEL
LIN {X 0,Y 235.269,Z 556.422,A -85,B 0,C 180,E1 -19751.94,E2 -19751.94} C_VEL
LIN {X 0,Y 234.954,Z 555.219,A -85,B 0,C 180,E1 -19752.725,E2 -19752.725} C_VEL
LIN {X 0,Y 234.96,Z 555.219,A -85,B 0,C 180,E1 -19756.53,E2 -19756.53} C_VEL
LIN {X 0,Y 234.953,Z 555.216,A -85,B 0,C 180,E1 -19761.085,E2 -19761.085} C_VEL
LIN {X 0,Y 234.958,Z 555.215,A -85,B 0,C 180,E1 -19765.366,E2 -19765.366} C_VEL
LIN {X 0,Y 234.966,Z 555.209,A -85,B 0,C 180,E1 -19770.156,E2 -19770.156} C_VEL
LIN {X 0,Y 234.991,Z 555.205,A -85,B 0,C 180,E1 -19773.793,E2 -19773.793} C_VEL
LIN {X 0,Y 235.008,Z 555.207,A -85,B 0,C 180,E1 -19778.969,E2 -19778.969} C_VEL
LIN {X 0,Y 235.092,Z 555.193,A -85,B 0,C 180,E1 -19783.059,E2 -19783.059} C_VEL
LIN {X 0,Y 235.109,Z 555.188,A -85,B 0,C 180,E1 -19787.921,E2 -19787.921} C_VEL
LIN {X 0,Y 235.326,Z 555.164,A -85,B 0,C 180,E1 -19791.412,E2 -19791.412} C_VEL
LIN {X 0,Y 235.368,Z 555.156,A -85,B 0,C 180,E1 -19793.14,E2 -19793.14} C_VEL
LIN {X 0,Y 235.591,Z 555.125,A -85,B 0,C 180,E1 -19798.29,E2 -19798.29} C_VEL
LIN {X 0,Y 235.59,Z 555.136,A -85,B 0,C 180,E1 -19801.709,E2 -19801.709} C_VEL
LIN {X 0,Y 235.368,Z 555.163,A -85,B 0,C 180,E1 -19806.86,E2 -19806.86} C_VEL
LIN {X 0,Y 235.209,Z 555.183,A -85,B 0,C 180,E1 -19810.328,E2 -19810.328} C_VEL
LIN {X 0,Y 235.107,Z 555.198,A -85,B 0,C 180,E1 -19815.607,E2 -19815.607} C_VEL
LIN {X 0,Y 235.003,Z 555.205,A -85,B 0,C 180,E1 -19819.206,E2 -19819.206} C_VEL
LIN {X 0,Y 234.971,Z 555.211,A -85,B 0,C 180,E1 -19821.788,E2 -19821.788} C_VEL
LIN {X 0,Y 234.288,Z 555.296,A -85,B 0,C 180,E1 -19823.22,E2 -19823.22} C_VEL
LIN {X 0,Y 231.372,Z 555.663,A -85,B 0,C 180,E1 -19825.554,E2 -19825.554} C_VEL
LIN {X 0,Y 228.936,Z 555.959,A -85,B 0,C 180,E1 -19827.458,E2 -19827.458} C_VEL
LIN {X 0,Y 227.952,Z 556.09,A -85,B 0,C 180,E1 -19828.938,E2 -19828.938} C_VEL
LIN {X 0,Y 227.905,Z 556.094,A -85,B 0,C 180,E1 -19829.438,E2 -19829.438} C_VEL
LIN {X 0,Y 227.886,Z 556.098,A -85,B 0,C 180,E1 -19833.719,E2 -19833.719} C_VEL
LIN {X 0,Y 227.868,Z 556.1,A -85,B 0,C 180,E1 -19838.086,E2 -19838.086} C_VEL
LIN {X 0,Y 227.863,Z 556.103,A -85,B 0,C 180,E1 -19842.73,E2 -19842.73} C_VEL
LIN {X 0,Y 227.865,Z 556.188,A -85,B 0,C 180,E1 -19845.575,E2 -19845.575} C_VEL
LIN {X 0,Y 230.074,Z 564.385,A -85,B 0,C 180,E1 -19850.099,E2 -19850.099} C_VEL
LIN {X 0,Y 230.669,Z 566.398,A -85,B 0,C 180,E1 -19851.153,E2 -19851.153} C_VEL
LIN {X 0,Y 232.867,Z 570.603,A -85,B 0,C 180,E1 -19851.779,E2 -19851.779} C_VEL
LIN {X 0,Y 238.702,Z 581.696,A -85,B 0,C 180,E1 -19853.357,E2 -19853.357} C_VEL
LIN {X 0,Y 245.741,Z 596.486,A -85,B 0,C 180,E1 -19855.17,E2 -19855.17} C_VEL
LIN {X 0,Y 249.48,Z 605.957,A -85,B 0,C 180,E1 -19856.131,E2 -19856.131} C_VEL
LIN {X 0,Y 251.791,Z 621.339,A -85,B 0,C 180,E1 -19857.029,E2 -19857.029} C_VEL
LIN {X 0,Y 249.504,Z 675.181,A -85,B 0,C 180,E1 -19858.546,E2 -19858.546} C_VEL
LIN {X 0,Y 248.159,Z 688.596,A -85,B 0,C 180,E1 -19859.204,E2 -19859.204} C_VEL
LIN {X 0,Y 246.228,Z 701.506,A -85,B 0,C 180,E1 -19860.152,E2 -19860.152} C_VEL
LIN {X 0,Y 243.969,Z 713.436,A -85,B 0,C 180,E1 -19861.386,E2 -19861.386} C_VEL
LIN {X 0,Y 241.394,Z 724.869,A -85,B 0,C 180,E1 -19862.942,E2 -19862.942} C_VEL
LIN {X 0,Y 238.647,Z 735.187,A -85,B 0,C 180,E1 -19864.722,E2 -19864.722} C_VEL
LIN {X 0,Y 235.891,Z 744.465,A -85,B 0,C 180,E1 -19866.749,E2 -19866.749} C_VEL
LIN {X 0,Y 233.391,Z 752.606,A -85,B 0,C 180,E1 -19868.985,E2 -19868.985} C_VEL
LIN {X 0,Y 231.202,Z 759.618,A -85,B 0,C 180,E1 -19871.387,E2 -19871.387} C_VEL
LIN {X 0,Y 229.219,Z 765.663,A -85,B 0,C 180,E1 -19873.982,E2 -19873.982} C_VEL
LIN {X 0,Y 227.686,Z 770.46,A -85,B 0,C 180,E1 -19876.615,E2 -19876.615} C_VEL
LIN {X 0,Y 226.657,Z 774.151,A -85,B 0,C 180,E1 -19879.278,E2 -19879.278} C_VEL
LIN {X 0,Y 226.16,Z 776.065,A -85,B 0,C 180,E1 -19881.062,E2 -19881.062} C_VEL
LIN {X 0,Y 225.826,Z 777.539,A -85,B 0,C 180,E1 -19882.849,E2 -19882.849} C_VEL
LIN {X 0,Y 225.59,Z 779.247,A -85,B 0,C 180,E1 -19886.428,E2 -19886.428} C_VEL
LIN {X 0,Y 225.662,Z 779.524,A -85,B 0,C 180,E1 -19888.215,E2 -19888.215} C_VEL
LIN {X 0,Y 225.736,Z 779.394,A -85,B 0,C 180,E1 -19890,E2 -19890} C_VEL
LIN {X 0,Y 225.667,Z 778.831,A -85,B 0,C 180,E1 -19891.785,E2 -19891.785} C_VEL
LIN {X 0,Y 225.664,Z 777.043,A -85,B 0,C 180,E1 -19894.727,E2 -19894.727} C_VEL
LIN {X 0,Y 225.953,Z 773.658,A -85,B 0,C 180,E1 -19898.046,E2 -19898.046} C_VEL
LIN {X 0,Y 226.531,Z 769.754,A -85,B 0,C 180,E1 -19900.728,E2 -19900.728} C_VEL
LIN {X 0,Y 227.455,Z 764.712,A -85,B 0,C 180,E1 -19903.399,E2 -19903.399} C_VEL
LIN {X 0,Y 228.98,Z 758.383,A -85,B 0,C 180,E1 -19906.035,E2 -19906.035} C_VEL
LIN {X 0,Y 230.875,Z 750.444,A -85,B 0,C 180,E1 -19908.64,E2 -19908.64} C_VEL
LIN {X 0,Y 232.612,Z 742.286,A -85,B 0,C 180,E1 -19910.807,E2 -19910.807} C_VEL
LIN {X 0,Y 234.713,Z 732.456,A -85,B 0,C 180,E1 -19912.908,E2 -19912.908} C_VEL
LIN {X 0,Y 237.003,Z 721.403,A -85,B 0,C 180,E1 -19914.762,E2 -19914.762} C_VEL
LIN {X 0,Y 238.884,Z 710.55,A -85,B 0,C 180,E1 -19916.186,E2 -19916.186} C_VEL
LIN {X 0,Y 240.696,Z 698.592,A -85,B 0,C 180,E1 -19917.379,E2 -19917.379} C_VEL
LIN {X 0,Y 242.196,Z 685.628,A -85,B 0,C 180,E1 -19918.31,E2 -19918.31} C_VEL
LIN {X 0,Y 243.124,Z 672.766,A -85,B 0,C 180,E1 -19918.9,E2 -19918.9} C_VEL
LIN {X 0,Y 245.073,Z 618.548,A -85,B 0,C 180,E1 -19920.446,E2 -19920.446} C_VEL
LIN {X 0,Y 241.797,Z 593.851,A -85,B 0,C 180,E1 -19921.691,E2 -19921.691} C_VEL
LIN {X 0,Y 235.348,Z 577.878,A -85,B 0,C 180,E1 -19923.146,E2 -19923.146} C_VEL
LIN {X 0,Y 230.463,Z 566.842,A -85,B 0,C 180,E1 -19924.286,E2 -19924.286} C_VEL
LIN {X 0,Y 228.622,Z 559.02,A -85,B 0,C 180,E1 -19927.937,E2 -19927.937} C_VEL
LIN {X 0,Y 227.875,Z 556.098,A -85,B 0,C 180,E1 -19929.398,E2 -19929.398} C_VEL
LIN {X 0,Y 227.814,Z 556.107,A -85,B 0,C 180,E1 -19932.74,E2 -19932.74} C_VEL
LIN {X 0,Y 227.863,Z 556.099,A -85,B 0,C 180,E1 -19937.27,E2 -19937.27} C_VEL
LIN {X 0,Y 227.868,Z 556.1,A -85,B 0,C 180,E1 -19941.914,E2 -19941.914} C_VEL
LIN {X 0,Y 227.887,Z 556.095,A -85,B 0,C 180,E1 -19946.373,E2 -19946.373} C_VEL
LIN {X 0,Y 227.915,Z 556.092,A -85,B 0,C 180,E1 -19950.437,E2 -19950.437} C_VEL
LIN {X 0,Y 227.921,Z 556.093,A -85,B 0,C 180,E1 -19954.425,E2 -19954.425} C_VEL
LIN {X 0,Y 227.943,Z 556.089,A -85,B 0,C 180,E1 -19958.285,E2 -19958.285} C_VEL
LIN {X 0,Y 228.029,Z 556.071,A -85,B 0,C 180,E1 -19962.827,E2 -19962.827} C_VEL
LIN {X 0,Y 228.068,Z 556.069,A -85,B 0,C 180,E1 -19967.543,E2 -19967.543} C_VEL
LIN {X 0,Y 228.3,Z 556.045,A -85,B 0,C 180,E1 -19971.146,E2 -19971.146} C_VEL
LIN {X 0,Y 228.348,Z 556.041,A -85,B 0,C 180,E1 -19972.929,E2 -19972.929} C_VEL
LIN {X 0,Y 228.549,Z 556.015,A -85,B 0,C 180,E1 -19978.238,E2 -19978.238} C_VEL
LIN {X 0,Y 228.549,Z 556.005,A -85,B 0,C 180,E1 -19981.762,E2 -19981.762} C_VEL
LIN {X 0,Y 228.334,Z 556.043,A -85,B 0,C 180,E1 -19987.072,E2 -19987.072} C_VEL
LIN {X 0,Y 228.141,Z 556.046,A -85,B 0,C 180,E1 -19990.652,E2 -19990.652} C_VEL
LIN {X 0,Y 228.058,Z 556.075,A -85,B 0,C 180,E1 -19994.273,E2 -19994.273} C_VEL
LIN {X 0,Y 227.999,Z 556.076,A -85,B 0,C 180,E1 -19997.954,E2 -19997.954} C_VEL
LIN {X 0,Y 227.927,Z 556.089,A -85,B 0,C 180,E1 -20002.33,E2 -20002.33} C_VEL
LIN {X 0,Y 227.94,Z 556.085,A -85,B 0,C 180,E1 -20006.604,E2 -20006.604} C_VEL
LIN {X 0,Y 227.906,Z 556.093,A -85,B 0,C 180,E1 -20010.297,E2 -20010.297} C_VEL
LIN {X 0,Y 227.887,Z 556.099,A -85,B 0,C 180,E1 -20013.719,E2 -20013.719} C_VEL
LIN {X 0,Y 227.858,Z 556.085,A -85,B 0,C 180,E1 -20018.089,E2 -20018.089} C_VEL
LIN {X 0,Y 227.864,Z 556.099,A -85,B 0,C 180,E1 -20022.731,E2 -20022.731} C_VEL
LIN {X 0,Y 227.909,Z 556.094,A -85,B 0,C 180,E1 -20027.739,E2 -20027.739} C_VEL
LIN {X 0,Y 227.871,Z 556.099,A -85,B 0,C 180,E1 -20031.915,E2 -20031.915} C_VEL
LIN {X 0,Y 227.891,Z 556.098,A -85,B 0,C 180,E1 -20036.374,E2 -20036.374} C_VEL
LIN {X 0,Y 227.911,Z 556.164,A -85,B 0,C 180,E1 -20039.358,E2 -20039.358} C_VEL
LIN {X 0,Y 229.056,Z 559.184,A -85,B 0,C 180,E1 -20039.677,E2 -20039.677} C_VEL
LIN {X 0,Y 230.403,Z 561.371,A -85,B 0,C 180,E1 -20039.971,E2 -20039.971} C_VEL
LIN {X 0,Y 235.54,Z 571.601,A -85,B 0,C 180,E1 -20041.12,E2 -20041.12} C_VEL
LIN {X 0,Y 241.682,Z 586.044,A -85,B 0,C 180,E1 -20042.488,E2 -20042.488} C_VEL
LIN {X 0,Y 245.823,Z 596.993,A -85,B 0,C 180,E1 -20043.402,E2 -20043.402} C_VEL
LIN {X 0,Y 243.898,Z 650.335,A -85,B 0,C 180,E1 -20044.901,E2 -20044.901} C_VEL
LIN {X 0,Y 243.179,Z 666.533,A -85,B 0,C 180,E1 -20045.453,E2 -20045.453} C_VEL
LIN {X 0,Y 242.197,Z 678.471,A -85,B 0,C 180,E1 -20046.145,E2 -20046.145} C_VEL
LIN {X 0,Y 240.668,Z 691.351,A -85,B 0,C 180,E1 -20047.237,E2 -20047.237} C_VEL
LIN {X 0,Y 238.768,Z 703.565,A -85,B 0,C 180,E1 -20048.639,E2 -20048.639} C_VEL
LIN {X 0,Y 236.839,Z 714.453,A -85,B 0,C 180,E1 -20050.273,E2 -20050.273} C_VEL
LIN {X 0,Y 234.748,Z 724.285,A -85,B 0,C 180,E1 -20052.13,E2 -20052.13} C_VEL
LIN {X 0,Y 232.552,Z 733.23,A -85,B 0,C 180,E1 -20054.218,E2 -20054.218} C_VEL
LIN {X 0,Y 230.734,Z 741.935,A -85,B 0,C 180,E1 -20056.795,E2 -20056.795} C_VEL
LIN {X 0,Y 229.056,Z 748.911,A -85,B 0,C 180,E1 -20059.392,E2 -20059.392} C_VEL
LIN {X 0,Y 227.84,Z 754.482,A -85,B 0,C 180,E1 -20062.021,E2 -20062.021} C_VEL
LIN {X 0,Y 226.733,Z 758.88,A -85,B 0,C 180,E1 -20064.664,E2 -20064.664} C_VEL
LIN {X 0,Y 226.267,Z 761.202,A -85,B 0,C 180,E1 -20066.439,E2 -20066.439} C_VEL
LIN {X 0,Y 225.975,Z 763.099,A -85,B 0,C 180,E1 -20068.218,E2 -20068.218} C_VEL
LIN {X 0,Y 225.798,Z 764.567,A -85,B 0,C 180,E1 -20070,E2 -20070} C_VEL
LIN {X 0,Y 225.711,Z 765.599,A -85,B 0,C 180,E1 -20071.784,E2 -20071.784} C_VEL
LIN {X 0,Y 225.633,Z 766.457,A -85,B 0,C 180,E1 -20074.626,E2 -20074.626} C_VEL
LIN {X 0,Y 225.722,Z 766.404,A -85,B 0,C 180,E1 -20077.154,E2 -20077.154} C_VEL
LIN {X 0,Y 226.201,Z 764.923,A -85,B 0,C 180,E1 -20080.744,E2 -20080.744} C_VEL
LIN {X 0,Y 226.628,Z 763.597,A -85,B 0,C 180,E1 -20082.537,E2 -20082.537} C_VEL
LIN {X 0,Y 227.646,Z 760.777,A -85,B 0,C 180,E1 -20085.213,E2 -20085.213} C_VEL
LIN {X 0,Y 229.034,Z 756.783,A -85,B 0,C 180,E1 -20087.963,E2 -20087.963} C_VEL
LIN {X 0,Y 230.674,Z 751.934,A -85,B 0,C 180,E1 -20090.51,E2 -20090.51} C_VEL
LIN {X 0,Y 232.831,Z 745.641,A -85,B 0,C 180,E1 -20093.104,E2 -20093.104} C_VEL
LIN {X 0,Y 235.521,Z 737.732,A -85,B 0,C 180,E1 -20095.637,E2 -20095.637} C_VEL
LIN {X 0,Y 237.817,Z 729.69,A -85,B 0,C 180,E1 -20097.728,E2 -20097.728} C_VEL
LIN {X 0,Y 240.559,Z 719.775,A -85,B 0,C 180,E1 -20099.778,E2 -20099.778} C_VEL
LIN {X 0,Y 242.986,Z 710.051,A -85,B 0,C 180,E1 -20101.373,E2 -20101.373} C_VEL
LIN {X 0,Y 245.283,Z 699.518,A -85,B 0,C 180,E1 -20102.739,E2 -20102.739} C_VEL
LIN {X 0,Y 247.336,Z 686.787,A -85,B 0,C 180,E1 -20104.015,E2 -20104.015} C_VEL
LIN {X 0,Y 249.07,Z 673.88,A -85,B 0,C 180,E1 -20104.919,E2 -20104.919} C_VEL
LIN {X 0,Y 250.075,Z 660.956,A -85,B 0,C 180,E1 -20105.515,E2 -20105.515} C_VEL
LIN {X 0,Y 252.421,Z 604.476,A -85,B 0,C 180,E1 -20107.09,E2 -20107.09} C_VEL
LIN {X 0,Y 246.393,Z 590.386,A -85,B 0,C 180,E1 -20108.58,E2 -20108.58} C_VEL
LIN {X 0,Y 238.933,Z 575.469,A -85,B 0,C 180,E1 -20110.478,E2 -20110.478} C_VEL
LIN {X 0,Y 232.31,Z 564.004,A -85,B 0,C 180,E1 -20112.242,E2 -20112.242} C_VEL
LIN {X 0,Y 229.954,Z 560.261,A -85,B 0,C 180,E1 -20112.893,E2 -20112.893} C_VEL
LIN {X 0,Y 228.375,Z 557.868,A -85,B 0,C 180,E1 -20113.335,E2 -20113.335} C_VEL
LIN {X 0,Y 228.022,Z 556.637,A -85,B 0,C 180,E1 -20113.502,E2 -20113.502} C_VEL
LIN {X 0,Y 227.914,Z 556.094,A -85,B 0,C 180,E1 -20113.879,E2 -20113.879} C_VEL
LIN {X 0,Y 227.896,Z 556.085,A -85,B 0,C 180,E1 -20117.741,E2 -20117.741} C_VEL
LIN {X 0,Y 227.869,Z 556.102,A -85,B 0,C 180,E1 -20121.913,E2 -20121.913} C_VEL
LIN {X 0,Y 227.888,Z 556.093,A -85,B 0,C 180,E1 -20126.372,E2 -20126.372} C_VEL
LIN {X 0,Y 227.916,Z 556.089,A -85,B 0,C 180,E1 -20130.437,E2 -20130.437} C_VEL
LIN {X 0,Y 227.926,Z 556.088,A -85,B 0,C 180,E1 -20134.425,E2 -20134.425} C_VEL
LIN {X 0,Y 227.958,Z 556.08,A -85,B 0,C 180,E1 -20138.286,E2 -20138.286} C_VEL
LIN {X 0,Y 228.031,Z 556.071,A -85,B 0,C 180,E1 -20142.825,E2 -20142.825} C_VEL
LIN {X 0,Y 228.067,Z 556.063,A -85,B 0,C 180,E1 -20147.543,E2 -20147.543} C_VEL
LIN {X 0,Y 228.262,Z 556.046,A -85,B 0,C 180,E1 -20151.144,E2 -20151.144} C_VEL
LIN {X 0,Y 228.319,Z 556.033,A -85,B 0,C 180,E1 -20152.927,E2 -20152.927} C_VEL
LIN {X 0,Y 228.55,Z 556.002,A -85,B 0,C 180,E1 -20158.238,E2 -20158.238} C_VEL
LIN {X 0,Y 228.549,Z 556.012,A -85,B 0,C 180,E1 -20161.762,E2 -20161.762} C_VEL
LIN {X 0,Y 228.319,Z 556.04,A -85,B 0,C 180,E1 -20167.072,E2 -20167.072} C_VEL
LIN {X 0,Y 228.141,Z 556.066,A -85,B 0,C 180,E1 -20170.651,E2 -20170.651} C_VEL
LIN {X 0,Y 228.057,Z 556.066,A -85,B 0,C 180,E1 -20174.272,E2 -20174.272} C_VEL
LIN {X 0,Y 227.998,Z 556.075,A -85,B 0,C 180,E1 -20177.954,E2 -20177.954} C_VEL
LIN {X 0,Y 227.912,Z 556.087,A -85,B 0,C 180,E1 -20182.321,E2 -20182.321} C_VEL
LIN {X 0,Y 227.939,Z 556.083,A -85,B 0,C 180,E1 -20186.603,E2 -20186.603} C_VEL
LIN {X 0,Y 227.905,Z 556.094,A -85,B 0,C 180,E1 -20189.438,E2 -20189.438} C_VEL
LIN {X 0,Y 227.331,Z 556.18,A -85,B 0,C 180,E1 -20190.913,E2 -20190.913} C_VEL
LIN {X 0,Y 225.8,Z 556.379,A -85,B 0,C 180,E1 -20192.363,E2 -20192.363} C_VEL
LIN {X 0,Y 222.058,Z 556.84,A -85,B 0,C 180,E1 -20195.284,E2 -20195.284} C_VEL
LIN {X 0,Y 220.947,Z 556.967,A -85,B 0,C 180,E1 -20196.809,E2 -20196.809} C_VEL
LIN {X 0,Y 220.833,Z 556.977,A -85,B 0,C 180,E1 -20197.327,E2 -20197.327} C_VEL
LIN {X 0,Y 220.836,Z 556.979,A -85,B 0,C 180,E1 -20200.202,E2 -20200.202} C_VEL
LIN {X 0,Y 220.797,Z 557.05,A -85,B 0,C 180,E1 -20204.239,E2 -20204.239} C_VEL
LIN {X 0,Y 222.829,Z 564.336,A -85,B 0,C 180,E1 -20208.523,E2 -20208.523} C_VEL
LIN {X 0,Y 223.31,Z 566.192,A -85,B 0,C 180,E1 -20209.511,E2 -20209.511} C_VEL
LIN {X 0,Y 225.479,Z 570.223,A -85,B 0,C 180,E1 -20210.176,E2 -20210.176} C_VEL
LIN {X 0,Y 226.859,Z 572.581,A -85,B 0,C 180,E1 -20210.581,E2 -20210.581} C_VEL
LIN {X 0,Y 232.009,Z 582.064,A -85,B 0,C 180,E1 -20212.055,E2 -20212.055} C_VEL
LIN {X 0,Y 239.122,Z 596.76,A -85,B 0,C 180,E1 -20213.999,E2 -20213.999} C_VEL
LIN {X 0,Y 243.885,Z 608.16,A -85,B 0,C 180,E1 -20215.267,E2 -20215.267} C_VEL
LIN {X 0,Y 245.952,Z 622.952,A -85,B 0,C 180,E1 -20216.142,E2 -20216.142} C_VEL
LIN {X 0,Y 243.592,Z 675.228,A -85,B 0,C 180,E1 -20217.642,E2 -20217.642} C_VEL
LIN {X 0,Y 242.116,Z 689.175,A -85,B 0,C 180,E1 -20218.348,E2 -20218.348} C_VEL
LIN {X 0,Y 240.117,Z 701.841,A -85,B 0,C 180,E1 -20219.312,E2 -20219.312} C_VEL
LIN {X 0,Y 237.779,Z 713.636,A -85,B 0,C 180,E1 -20220.569,E2 -20220.569} C_VEL
LIN {X 0,Y 235.109,Z 724.995,A -85,B 0,C 180,E1 -20222.156,E2 -20222.156} C_VEL
LIN {X 0,Y 232.239,Z 735.251,A -85,B 0,C 180,E1 -20223.973,E2 -20223.973} C_VEL
LIN {X 0,Y 229.383,Z 744.468,A -85,B 0,C 180,E1 -20226.049,E2 -20226.049} C_VEL
LIN {X 0,Y 226.582,Z 753.125,A -85,B 0,C 180,E1 -20228.516,E2 -20228.516} C_VEL
LIN {X 0,Y 224.104,Z 760.675,A -85,B 0,C 180,E1 -20231.25,E2 -20231.25} C_VEL
LIN {X 0,Y 222.386,Z 765.573,A -85,B 0,C 180,E1 -20233.476,E2 -20233.476} C_VEL
LIN {X 0,Y 220.738,Z 770.345,A -85,B 0,C 180,E1 -20236.185,E2 -20236.185} C_VEL
LIN {X 0,Y 219.663,Z 774.013,A -85,B 0,C 180,E1 -20238.933,E2 -20238.933} C_VEL
LIN {X 0,Y 219.114,Z 775.916,A -85,B 0,C 180,E1 -20240.772,E2 -20240.772} C_VEL
LIN {X 0,Y 218.764,Z 777.37,A -85,B 0,C 180,E1 -20242.617,E2 -20242.617} C_VEL
LIN {X 0,Y 218.498,Z 779.057,A -85,B 0,C 180,E1 -20246.312,E2 -20246.312} C_VEL
LIN {X 0,Y 218.558,Z 779.324,A -85,B 0,C 180,E1 -20248.157,E2 -20248.157} C_VEL
LIN {X 0,Y 218.65,Z 779.174,A -85,B 0,C 180,E1 -20250,E2 -20250} C_VEL
LIN {X 0,Y 218.564,Z 778.601,A -85,B 0,C 180,E1 -20251.843,E2 -20251.843} C_VEL
LIN {X 0,Y 218.551,Z 777.07,A -85,B 0,C 180,E1 -20254.53,E2 -20254.53} C_VEL
LIN {X 0,Y 218.893,Z 773.384,A -85,B 0,C 180,E1 -20258.307,E2 -20258.307} C_VEL
LIN {X 0,Y 219.522,Z 769.457,A -85,B 0,C 180,E1 -20261.075,E2 -20261.075} C_VEL
LIN {X 0,Y 220.523,Z 764.39,A -85,B 0,C 180,E1 -20263.829,E2 -20263.829} C_VEL
LIN {X 0,Y 222.152,Z 758.027,A -85,B 0,C 180,E1 -20266.542,E2 -20266.542} C_VEL
LIN {X 0,Y 224.132,Z 750.048,A -85,B 0,C 180,E1 -20269.222,E2 -20269.222} C_VEL
LIN {X 0,Y 225.9,Z 742.082,A -85,B 0,C 180,E1 -20271.394,E2 -20271.394} C_VEL
LIN {X 0,Y 228.169,Z 731.976,A -85,B 0,C 180,E1 -20273.604,E2 -20273.604} C_VEL
LIN {X 0,Y 230.551,Z 720.831,A -85,B 0,C 180,E1 -20275.504,E2 -20275.504} C_VEL
LIN {X 0,Y 232.507,Z 709.889,A -85,B 0,C 180,E1 -20276.962,E2 -20276.962} C_VEL
LIN {X 0,Y 234.378,Z 697.803,A -85,B 0,C 180,E1 -20278.181,E2 -20278.181} C_VEL
LIN {X 0,Y 235.863,Z 685.4,A -85,B 0,C 180,E1 -20279.081,E2 -20279.081} C_VEL
LIN {X 0,Y 236.835,Z 672.523,A -85,B 0,C 180,E1 -20279.682,E2 -20279.682} C_VEL
LIN {X 0,Y 238.852,Z 619.479,A -85,B 0,C 180,E1 -20281.225,E2 -20281.225} C_VEL
LIN {X 0,Y 235.781,Z 596.171,A -85,B 0,C 180,E1 -20282.447,E2 -20282.447} C_VEL
LIN {X 0,Y 229.85,Z 581.308,A -85,B 0,C 180,E1 -20283.852,E2 -20283.852} C_VEL
LIN {X 0,Y 224.477,Z 569.684,A -85,B 0,C 180,E1 -20285.141,E2 -20285.141} C_VEL
LIN {X 0,Y 223.188,Z 566.524,A -85,B 0,C 180,E1 -20285.518,E2 -20285.518} C_VEL
LIN {X 0,Y 221.206,Z 558.554,A -85,B 0,C 180,E1 -20289.45,E2 -20289.45} C_VEL
LIN {X 0,Y 220.801,Z 556.981,A -85,B 0,C 180,E1 -20290.33,E2 -20290.33} C_VEL
LIN {X 0,Y 220.802,Z 556.981,A -85,B 0,C 180,E1 -20295.553,E2 -20295.553} C_VEL
LIN {X 0,Y 220.847,Z 556.973,A -85,B 0,C 180,E1 -20300.472,E2 -20300.472} C_VEL
LIN {X 0,Y 220.812,Z 556.979,A -85,B 0,C 180,E1 -20305.047,E2 -20305.047} C_VEL
LIN {X 0,Y 220.865,Z 556.974,A -85,B 0,C 180,E1 -20309.394,E2 -20309.394} C_VEL
LIN {X 0,Y 220.891,Z 556.969,A -85,B 0,C 180,E1 -20313.549,E2 -20313.549} C_VEL
LIN {X 0,Y 220.861,Z 556.967,A -85,B 0,C 180,E1 -20317.552,E2 -20317.552} C_VEL
LIN {X 0,Y 220.979,Z 556.948,A -85,B 0,C 180,E1 -20322.572,E2 -20322.572} C_VEL
LIN {X 0,Y 221.006,Z 556.952,A -85,B 0,C 180,E1 -20327.138,E2 -20327.138} C_VEL
LIN {X 0,Y 221.231,Z 556.924,A -85,B 0,C 180,E1 -20330.861,E2 -20330.861} C_VEL
LIN {X 0,Y 221.283,Z 556.92,A -85,B 0,C 180,E1 -20332.702,E2 -20332.702} C_VEL
LIN {X 0,Y 221.507,Z 556.892,A -85,B 0,C 180,E1 -20338.182,E2 -20338.182} C_VEL
LIN {X 0,Y 221.507,Z 556.881,A -85,B 0,C 180,E1 -20341.818,E2 -20341.818} C_VEL
LIN {X 0,Y 221.267,Z 556.922,A -85,B 0,C 180,E1 -20347.299,E2 -20347.299} C_VEL
LIN {X 0,Y 221.063,Z 556.927,A -85,B 0,C 180,E1 -20350.997,E2 -20350.997} C_VEL
LIN {X 0,Y 221.012,Z 556.953,A -85,B 0,C 180,E1 -20356.63,E2 -20356.63} C_VEL
LIN {X 0,Y 220.889,Z 556.952,A -85,B 0,C 180,E1 -20360.487,E2 -20360.487} C_VEL
LIN {X 0,Y 220.864,Z 556.972,A -85,B 0,C 180,E1 -20364.436,E2 -20364.436} C_VEL
LIN {X 0,Y 220.834,Z 556.975,A -85,B 0,C 180,E1 -20368.514,E2 -20368.514} C_VEL
LIN {X 0,Y 220.822,Z 556.976,A -85,B 0,C 180,E1 -20372.756,E2 -20372.756} C_VEL
LIN {X 0,Y 220.837,Z 556.958,A -85,B 0,C 180,E1 -20377.289,E2 -20377.289} C_VEL
LIN {X 0,Y 220.812,Z 556.978,A -85,B 0,C 180,E1 -20381.943,E2 -20381.943} C_VEL
LIN {X 0,Y 220.866,Z 556.971,A -85,B 0,C 180,E1 -20387.044,E2 -20387.044} C_VEL
LIN {X 0,Y 220.856,Z 556.972,A -85,B 0,C 180,E1 -20390.475,E2 -20390.475} C_VEL
LIN {X 0,Y 220.816,Z 556.98,A -85,B 0,C 180,E1 -20395.049,E2 -20395.049} C_VEL
LIN {X 0,Y 220.822,Z 557.002,A -85,B 0,C 180,E1 -20398.209,E2 -20398.209} C_VEL
LIN {X 0,Y 221.89,Z 559.912,A -85,B 0,C 180,E1 -20398.507,E2 -20398.507} C_VEL
LIN {X 0,Y 223.632,Z 562.731,A -85,B 0,C 180,E1 -20398.913,E2 -20398.913} C_VEL
LIN {X 0,Y 228.378,Z 571.388,A -85,B 0,C 180,E1 -20400.014,E2 -20400.014} C_VEL
LIN {X 0,Y 235.359,Z 587.445,A -85,B 0,C 180,E1 -20401.647,E2 -20401.647} C_VEL
LIN {X 0,Y 239.543,Z 598.588,A -85,B 0,C 180,E1 -20402.619,E2 -20402.619} C_VEL
LIN {X 0,Y 237.616,Z 650.644,A -85,B 0,C 180,E1 -20404.119,E2 -20404.119} C_VEL
LIN {X 0,Y 236.851,Z 666.95,A -85,B 0,C 180,E1 -20404.689,E2 -20404.689} C_VEL
LIN {X 0,Y 235.77,Z 679.533,A -85,B 0,C 180,E1 -20405.452,E2 -20405.452} C_VEL
LIN {X 0,Y 234.156,Z 692.178,A -85,B 0,C 180,E1 -20406.567,E2 -20406.567} C_VEL
LIN {X 0,Y 232.205,Z 704.263,A -85,B 0,C 180,E1 -20408.004,E2 -20408.004} C_VEL
LIN {X 0,Y 230.209,Z 715.024,A -85,B 0,C 180,E1 -20409.68,E2 -20409.68} C_VEL
LIN {X 0,Y 228.04,Z 724.793,A -85,B 0,C 180,E1 -20411.586,E2 -20411.586} C_VEL
LIN {X 0,Y 225.754,Z 733.688,A -85,B 0,C 180,E1 -20413.729,E2 -20413.729} C_VEL
LIN {X 0,Y 223.853,Z 742.348,A -85,B 0,C 180,E1 -20416.381,E2 -20416.381} C_VEL
LIN {X 0,Y 222.091,Z 749.273,A -85,B 0,C 180,E1 -20419.055,E2 -20419.055} C_VEL
LIN {X 0,Y 220.846,Z 754.812,A -85,B 0,C 180,E1 -20421.767,E2 -20421.767} C_VEL
LIN {X 0,Y 219.68,Z 759.182,A -85,B 0,C 180,E1 -20424.493,E2 -20424.493} C_VEL
LIN {X 0,Y 219.194,Z 761.49,A -85,B 0,C 180,E1 -20426.323,E2 -20426.323} C_VEL
LIN {X 0,Y 218.912,Z 763.373,A -85,B 0,C 180,E1 -20428.16,E2 -20428.16} C_VEL
LIN {X 0,Y 218.71,Z 764.815,A -85,B 0,C 180,E1 -20430,E2 -20430} C_VEL
LIN {X 0,Y 218.625,Z 765.835,A -85,B 0,C 180,E1 -20431.842,E2 -20431.842} C_VEL
LIN {X 0,Y 218.542,Z 766.643,A -85,B 0,C 180,E1 -20434.496,E2 -20434.496} C_VEL
LIN {X 0,Y 218.637,Z 766.592,A -85,B 0,C 180,E1 -20437.387,E2 -20437.387} C_VEL
LIN {X 0,Y 218.869,Z 766.03,A -85,B 0,C 180,E1 -20439.239,E2 -20439.239} C_VEL
LIN {X 0,Y 219.644,Z 763.746,A -85,B 0,C 180,E1 -20442.943,E2 -20442.943} C_VEL
LIN {X 0,Y 220.747,Z 760.899,A -85,B 0,C 180,E1 -20445.701,E2 -20445.701} C_VEL
LIN {X 0,Y 222.163,Z 757.02,A -85,B 0,C 180,E1 -20448.442,E2 -20448.442} C_VEL
LIN {X 0,Y 223.987,Z 751.997,A -85,B 0,C 180,E1 -20451.151,E2 -20451.151} C_VEL
LIN {X 0,Y 226.248,Z 745.659,A -85,B 0,C 180,E1 -20453.817,E2 -20453.817} C_VEL
LIN {X 0,Y 229.074,Z 737.703,A -85,B 0,C 180,E1 -20456.414,E2 -20456.414} C_VEL
LIN {X 0,Y 231.413,Z 729.938,A -85,B 0,C 180,E1 -20458.475,E2 -20458.475} C_VEL
LIN {X 0,Y 234.068,Z 720.716,A -85,B 0,C 180,E1 -20460.442,E2 -20460.442} C_VEL
LIN {X 0,Y 236.905,Z 709.837,A -85,B 0,C 180,E1 -20462.274,E2 -20462.274} C_VEL
LIN {X 0,Y 239.31,Z 699.167,A -85,B 0,C 180,E1 -20463.663,E2 -20463.663} C_VEL
LIN {X 0,Y 241.469,Z 686.28,A -85,B 0,C 180,E1 -20464.959,E2 -20464.959} C_VEL
LIN {X 0,Y 243.209,Z 673.387,A -85,B 0,C 180,E1 -20465.862,E2 -20465.862} C_VEL
LIN {X 0,Y 244.175,Z 661.148,A -85,B 0,C 180,E1 -20466.429,E2 -20466.429} C_VEL
LIN {X 0,Y 246.546,Z 606.405,A -85,B 0,C 180,E1 -20467.986,E2 -20467.986} C_VEL
LIN {X 0,Y 239.978,Z 591.284,A -85,B 0,C 180,E1 -20469.691,E2 -20469.691} C_VEL
LIN {X 0,Y 232.978,Z 577.525,A -85,B 0,C 180,E1 -20471.571,E2 -20471.571} C_VEL
LIN {X 0,Y 226.255,Z 565.852,A -85,B 0,C 180,E1 -20473.477,E2 -20473.477} C_VEL
LIN {X 0,Y 223.974,Z 562.503,A -85,B 0,C 180,E1 -20474.137,E2 -20474.137} C_VEL
LIN {X 0,Y 223.126,Z 561.367,A -85,B 0,C 180,E1 -20474.383,E2 -20474.383} C_VEL
LIN {X 0,Y 221.362,Z 558.944,A -85,B 0,C 180,E1 -20474.907,E2 -20474.907} C_VEL
LIN {X 0,Y 220.838,Z 556.974,A -85,B 0,C 180,E1 -20475.137,E2 -20475.137} C_VEL
LIN {X 0,Y 220.836,Z 556.961,A -85,B 0,C 180,E1 -20478.062,E2 -20478.062} C_VEL
LIN {X 0,Y 220.832,Z 556.973,A -85,B 0,C 180,E1 -20482.794,E2 -20482.794} C_VEL
LIN {X 0,Y 220.822,Z 556.977,A -85,B 0,C 180,E1 -20487.244,E2 -20487.244} C_VEL
LIN {X 0,Y 220.834,Z 556.977,A -85,B 0,C 180,E1 -20491.486,E2 -20491.486} C_VEL
LIN {X 0,Y 220.864,Z 556.973,A -85,B 0,C 180,E1 -20495.564,E2 -20495.564} C_VEL
LIN {X 0,Y 220.889,Z 556.97,A -85,B 0,C 180,E1 -20499.513,E2 -20499.513} C_VEL
LIN {X 0,Y 221.012,Z 556.948,A -85,B 0,C 180,E1 -20503.37,E2 -20503.37} C_VEL
LIN {X 0,Y 221.007,Z 556.943,A -85,B 0,C 180,E1 -20507.138,E2 -20507.138} C_VEL
LIN {X 0,Y 221.2,Z 556.927,A -85,B 0,C 180,E1 -20510.859,E2 -20510.859} C_VEL
LIN {X 0,Y 221.254,Z 556.912,A -85,B 0,C 180,E1 -20512.7,E2 -20512.7} C_VEL
LIN {X 0,Y 221.508,Z 556.879,A -85,B 0,C 180,E1 -20518.182,E2 -20518.182} C_VEL
LIN {X 0,Y 221.507,Z 556.888,A -85,B 0,C 180,E1 -20521.818,E2 -20521.818} C_VEL
LIN {X 0,Y 221.254,Z 556.919,A -85,B 0,C 180,E1 -20527.299,E2 -20527.299} C_VEL
LIN {X 0,Y 221.076,Z 556.948,A -85,B 0,C 180,E1 -20530.996,E2 -20530.996} C_VEL
LIN {X 0,Y 221.011,Z 556.954,A -85,B 0,C 180,E1 -20536.63,E2 -20536.63} C_VEL
LIN {X 0,Y 220.88,Z 556.972,A -85,B 0,C 180,E1 -20540.487,E2 -20540.487} C_VEL
LIN {X 0,Y 220.858,Z 556.971,A -85,B 0,C 180,E1 -20544.436,E2 -20544.436} C_VEL
LIN {X 0,Y 220.833,Z 556.972,A -85,B 0,C 180,E1 -20548.514,E2 -20548.514} C_VEL
LIN {X 0,Y 220.821,Z 556.978,A -85,B 0,C 180,E1 -20552.755,E2 -20552.755} C_VEL
LIN {X 0,Y 220.833,Z 556.977,A -85,B 0,C 180,E1 -20557.327,E2 -20557.327} C_VEL
LIN {X 0,Y 220.101,Z 557.069,A -85,B 0,C 180,E1 -20558.341,E2 -20558.341} C_VEL
LIN {X 0,Y 217.219,Z 557.428,A -85,B 0,C 180,E1 -20559.932,E2 -20559.932} C_VEL
LIN {X 0,Y 214.395,Z 557.781,A -85,B 0,C 180,E1 -20561.566,E2 -20561.566} C_VEL
LIN {X 0,Y 213.788,Z 557.856,A -85,B 0,C 180,E1 -20562.624,E2 -20562.624} C_VEL
LIN {X 0,Y 214.141,Z 559.455,A -85,B 0,C 180,E1 -20563.779,E2 -20563.779} C_VEL
LIN {X 0,Y 215.97,Z 565.833,A -85,B 0,C 180,E1 -20567.705,E2 -20567.705} C_VEL
LIN {X 0,Y 218.352,Z 570.157,A -85,B 0,C 180,E1 -20568.497,E2 -20568.497} C_VEL
LIN {X 0,Y 222.719,Z 577.691,A -85,B 0,C 180,E1 -20569.862,E2 -20569.862} C_VEL
LIN {X 0,Y 228.434,Z 588.385,A -85,B 0,C 180,E1 -20571.564,E2 -20571.564} C_VEL
LIN {X 0,Y 236.055,Z 604.957,A -85,B 0,C 180,E1 -20573.733,E2 -20573.733} C_VEL
LIN {X 0,Y 238.509,Z 611.66,A -85,B 0,C 180,E1 -20574.439,E2 -20574.439} C_VEL
LIN {X 0,Y 240.157,Z 624.232,A -85,B 0,C 180,E1 -20575.197,E2 -20575.197} C_VEL
LIN {X 0,Y 237.71,Z 675.441,A -85,B 0,C 180,E1 -20576.697,E2 -20576.697} C_VEL
LIN {X 0,Y 236.207,Z 689.143,A -85,B 0,C 180,E1 -20577.409,E2 -20577.409} C_VEL
LIN {X 0,Y 234.282,Z 701.127,A -85,B 0,C 180,E1 -20578.335,E2 -20578.335} C_VEL
LIN {X 0,Y 231.971,Z 712.262,A -85,B 0,C 180,E1 -20579.505,E2 -20579.505} C_VEL
LIN {X 0,Y 229.206,Z 723.833,A -85,B 0,C 180,E1 -20581.124,E2 -20581.124} C_VEL
LIN {X 0,Y 226.196,Z 734.258,A -85,B 0,C 180,E1 -20582.974,E2 -20582.974} C_VEL
LIN {X 0,Y 223.459,Z 742.788,A -85,B 0,C 180,E1 -20584.876,E2 -20584.876} C_VEL
LIN {X 0,Y 220.832,Z 750.665,A -85,B 0,C 180,E1 -20587.055,E2 -20587.055} C_VEL
LIN {X 0,Y 218.204,Z 758.376,A -85,B 0,C 180,E1 -20589.743,E2 -20589.743} C_VEL
LIN {X 0,Y 215.578,Z 765.484,A -85,B 0,C 180,E1 -20592.938,E2 -20592.938} C_VEL
LIN {X 0,Y 213.815,Z 770.231,A -85,B 0,C 180,E1 -20595.729,E2 -20595.729} C_VEL
LIN {X 0,Y 212.685,Z 773.876,A -85,B 0,C 180,E1 -20598.565,E2 -20598.565} C_VEL
LIN {X 0,Y 212.087,Z 775.767,A -85,B 0,C 180,E1 -20600.463,E2 -20600.463} C_VEL
LIN {X 0,Y 211.694,Z 777.2,A -85,B 0,C 180,E1 -20602.369,E2 -20602.369} C_VEL
LIN {X 0,Y 211.39,Z 778.783,A -85,B 0,C 180,E1 -20605.866,E2 -20605.866} C_VEL
LIN {X 0,Y 211.457,Z 779.124,A -85,B 0,C 180,E1 -20608.095,E2 -20608.095} C_VEL
LIN {X 0,Y 211.565,Z 778.955,A -85,B 0,C 180,E1 -20610,E2 -20610} C_VEL
LIN {X 0,Y 211.464,Z 778.37,A -85,B 0,C 180,E1 -20611.905,E2 -20611.905} C_VEL
LIN {X 0,Y 211.473,Z 777.008,A -85,B 0,C 180,E1 -20614.434,E2 -20614.434} C_VEL
LIN {X 0,Y 211.686,Z 774.185,A -85,B 0,C 180,E1 -20617.631,E2 -20617.631} C_VEL
LIN {X 0,Y 212.246,Z 770.598,A -85,B 0,C 180,E1 -20620.493,E2 -20620.493} C_VEL
LIN {X 0,Y 213.161,Z 765.892,A -85,B 0,C 180,E1 -20623.343,E2 -20623.343} C_VEL
LIN {X 0,Y 214.993,Z 758.814,A -85,B 0,C 180,E1 -20626.62,E2 -20626.62} C_VEL
LIN {X 0,Y 217.029,Z 751.139,A -85,B 0,C 180,E1 -20629.385,E2 -20629.385} C_VEL
LIN {X 0,Y 218.892,Z 743.269,A -85,B 0,C 180,E1 -20631.667,E2 -20631.667} C_VEL
LIN {X 0,Y 221.13,Z 733.647,A -85,B 0,C 180,E1 -20633.904,E2 -20633.904} C_VEL
LIN {X 0,Y 223.549,Z 722.984,A -85,B 0,C 180,E1 -20635.861,E2 -20635.861} C_VEL
LIN {X 0,Y 225.609,Z 712.685,A -85,B 0,C 180,E1 -20637.353,E2 -20637.353} C_VEL
LIN {X 0,Y 227.681,Z 700.428,A -85,B 0,C 180,E1 -20638.709,E2 -20638.709} C_VEL
LIN {X 0,Y 229.337,Z 687.513,A -85,B 0,C 180,E1 -20639.739,E2 -20639.739} C_VEL
LIN {X 0,Y 230.444,Z 675.055,A -85,B 0,C 180,E1 -20640.402,E2 -20640.402} C_VEL
LIN {X 0,Y 232.649,Z 620.15,A -85,B 0,C 180,E1 -20642.059,E2 -20642.059} C_VEL
LIN {X 0,Y 229.854,Z 598.599,A -85,B 0,C 180,E1 -20643.231,E2 -20643.231} C_VEL
LIN {X 0,Y 224.377,Z 584.786,A -85,B 0,C 180,E1 -20644.594,E2 -20644.594} C_VEL
LIN {X 0,Y 217.667,Z 570.124,A -85,B 0,C 180,E1 -20646.299,E2 -20646.299} C_VEL
LIN {X 0,Y 215.941,Z 566.327,A -85,B 0,C 180,E1 -20646.786,E2 -20646.786} C_VEL
LIN {X 0,Y 213.726,Z 557.859,A -85,B 0,C 180,E1 -20651.277,E2 -20651.277} C_VEL
LIN {X 0,Y 213.774,Z 557.853,A -85,B 0,C 180,E1 -20656.339,E2 -20656.339} C_VEL
LIN {X 0,Y 213.776,Z 557.857,A -85,B 0,C 180,E1 -20661.345,E2 -20661.345} C_VEL
LIN {X 0,Y 213.766,Z 557.855,A -85,B 0,C 180,E1 -20666.02,E2 -20666.02} C_VEL
LIN {X 0,Y 213.777,Z 557.853,A -85,B 0,C 180,E1 -20670.454,E2 -20670.454} C_VEL
LIN {X 0,Y 213.795,Z 557.853,A -85,B 0,C 180,E1 -20674.701,E2 -20674.701} C_VEL
LIN {X 0,Y 213.798,Z 557.851,A -85,B 0,C 180,E1 -20678.802,E2 -20678.802} C_VEL
LIN {X 0,Y 213.938,Z 557.825,A -85,B 0,C 180,E1 -20682.803,E2 -20682.803} C_VEL
LIN {X 0,Y 213.947,Z 557.833,A -85,B 0,C 180,E1 -20686.706,E2 -20686.706} C_VEL
LIN {X 0,Y 214.162,Z 557.804,A -85,B 0,C 180,E1 -20690.556,E2 -20690.556} C_VEL
LIN {X 0,Y 214.222,Z 557.799,A -85,B 0,C 180,E1 -20692.46,E2 -20692.46} C_VEL
LIN {X 0,Y 214.44,Z 557.772,A -85,B 0,C 180,E1 -20698.122,E2 -20698.122} C_VEL
LIN {X 0,Y 214.545,Z 557.758,A -85,B 0,C 180,E1 -20700,E2 -20700} C_VEL
LIN {X 0,Y 214.441,Z 557.761,A -85,B 0,C 180,E1 -20701.878,E2 -20701.878} C_VEL
LIN {X 0,Y 214.204,Z 557.799,A -85,B 0,C 180,E1 -20707.542,E2 -20707.542} C_VEL
LIN {X 0,Y 213.995,Z 557.807,A -85,B 0,C 180,E1 -20711.365,E2 -20711.365} C_VEL
LIN {X 0,Y 213.928,Z 557.837,A -85,B 0,C 180,E1 -20715.238,E2 -20715.238} C_VEL
LIN {X 0,Y 213.836,Z 557.83,A -85,B 0,C 180,E1 -20719.188,E2 -20719.188} C_VEL
LIN {X 0,Y 213.844,Z 557.846,A -85,B 0,C 180,E1 -20723.228,E2 -20723.228} C_VEL
LIN {X 0,Y 213.826,Z 557.845,A -85,B 0,C 180,E1 -20727.451,E2 -20727.451} C_VEL
LIN {X 0,Y 213.777,Z 557.851,A -85,B 0,C 180,E1 -20731.736,E2 -20731.736} C_VEL
LIN {X 0,Y 213.748,Z 557.848,A -85,B 0,C 180,E1 -20736.288,E2 -20736.288} C_VEL
LIN {X 0,Y 213.737,Z 557.861,A -85,B 0,C 180,E1 -20741.12,E2 -20741.12} C_VEL
LIN {X 0,Y 213.774,Z 557.855,A -85,B 0,C 180,E1 -20743.677,E2 -20743.677} C_VEL
LIN {X 0,Y 213.811,Z 557.848,A -85,B 0,C 180,E1 -20746.35,E2 -20746.35} C_VEL
LIN {X 0,Y 213.795,Z 557.85,A -85,B 0,C 180,E1 -20749.12,E2 -20749.12} C_VEL
LIN {X 0,Y 213.755,Z 557.856,A -85,B 0,C 180,E1 -20753.715,E2 -20753.715} C_VEL
LIN {X 0,Y 213.784,Z 557.857,A -85,B 0,C 180,E1 -20756.951,E2 -20756.951} C_VEL
LIN {X 0,Y 214.785,Z 560.708,A -85,B 0,C 180,E1 -20757.257,E2 -20757.257} C_VEL
LIN {X 0,Y 216.33,Z 563.07,A -85,B 0,C 180,E1 -20757.638,E2 -20757.638} C_VEL
LIN {X 0,Y 221.89,Z 572.846,A -85,B 0,C 180,E1 -20759,E2 -20759} C_VEL
LIN {X 0,Y 227.815,Z 585.86,A -85,B 0,C 180,E1 -20760.453,E2 -20760.453} C_VEL
LIN {X 0,Y 233.416,Z 600.525,A -85,B 0,C 180,E1 -20761.822,E2 -20761.822} C_VEL
LIN {X 0,Y 230.844,Z 663.104,A -85,B 0,C 180,E1 -20763.689,E2 -20763.689} C_VEL
LIN {X 0,Y 229.794,Z 676.417,A -85,B 0,C 180,E1 -20764.42,E2 -20764.42} C_VEL
LIN {X 0,Y 228.311,Z 688.938,A -85,B 0,C 180,E1 -20765.446,E2 -20765.446} C_VEL
LIN {X 0,Y 226.547,Z 700.232,A -85,B 0,C 180,E1 -20766.701,E2 -20766.701} C_VEL
LIN {X 0,Y 224.381,Z 711.846,A -85,B 0,C 180,E1 -20768.406,E2 -20768.406} C_VEL
LIN {X 0,Y 222.099,Z 722.284,A -85,B 0,C 180,E1 -20770.354,E2 -20770.354} C_VEL
LIN {X 0,Y 219.865,Z 730.831,A -85,B 0,C 180,E1 -20772.322,E2 -20772.322} C_VEL
LIN {X 0,Y 217.958,Z 738.689,A -85,B 0,C 180,E1 -20774.573,E2 -20774.573} C_VEL
LIN {X 0,Y 216.359,Z 745.203,A -85,B 0,C 180,E1 -20776.857,E2 -20776.857} C_VEL
LIN {X 0,Y 214.569,Z 752.166,A -85,B 0,C 180,E1 -20779.898,E2 -20779.898} C_VEL
LIN {X 0,Y 213.37,Z 756.739,A -85,B 0,C 180,E1 -20782.429,E2 -20782.429} C_VEL
LIN {X 0,Y 212.441,Z 760.708,A -85,B 0,C 180,E1 -20785.256,E2 -20785.256} C_VEL
LIN {X 0,Y 211.828,Z 763.647,A -85,B 0,C 180,E1 -20788.099,E2 -20788.099} C_VEL
LIN {X 0,Y 211.623,Z 765.064,A -85,B 0,C 180,E1 -20790,E2 -20790} C_VEL
LIN {X 0,Y 211.522,Z 766.071,A -85,B 0,C 180,E1 -20791.904,E2 -20791.904} C_VEL
LIN {X 0,Y 211.448,Z 766.824,A -85,B 0,C 180,E1 -20794.338,E2 -20794.338} C_VEL
LIN {X 0,Y 211.579,Z 766.778,A -85,B 0,C 180,E1 -20797.635,E2 -20797.635} C_VEL
LIN {X 0,Y 212.169,Z 765.246,A -85,B 0,C 180,E1 -20801.463,E2 -20801.463} C_VEL
LIN {X 0,Y 212.671,Z 763.894,A -85,B 0,C 180,E1 -20803.375,E2 -20803.375} C_VEL
LIN {X 0,Y 213.853,Z 761.022,A -85,B 0,C 180,E1 -20806.221,E2 -20806.221} C_VEL
LIN {X 0,Y 215.382,Z 757.114,A -85,B 0,C 180,E1 -20809.044,E2 -20809.044} C_VEL
LIN {X 0,Y 217.31,Z 752.06,A -85,B 0,C 180,E1 -20811.834,E2 -20811.834} C_VEL
LIN {X 0,Y 219.713,Z 745.672,A -85,B 0,C 180,E1 -20814.571,E2 -20814.571} C_VEL
LIN {X 0,Y 222.652,Z 737.674,A -85,B 0,C 180,E1 -20817.238,E2 -20817.238} C_VEL
LIN {X 0,Y 225.307,Z 729.381,A -85,B 0,C 180,E1 -20819.459,E2 -20819.459} C_VEL
LIN {X 0,Y 228.249,Z 719.511,A -85,B 0,C 180,E1 -20821.563,E2 -20821.563} C_VEL
LIN {X 0,Y 230.913,Z 709.609,A -85,B 0,C 180,E1 -20823.218,E2 -20823.218} C_VEL
LIN {X 0,Y 233.39,Z 698.819,A -85,B 0,C 180,E1 -20824.636,E2 -20824.636} C_VEL
LIN {X 0,Y 235.466,Z 686.915,A -85,B 0,C 180,E1 -20825.855,E2 -20825.855} C_VEL
LIN {X 0,Y 237.293,Z 673.981,A -85,B 0,C 180,E1 -20826.789,E2 -20826.789} C_VEL
LIN {X 0,Y 238.346,Z 661.687,A -85,B 0,C 180,E1 -20827.374,E2 -20827.374} C_VEL
LIN {X 0,Y 240.761,Z 608.462,A -85,B 0,C 180,E1 -20828.917,E2 -20828.917} C_VEL
LIN {X 0,Y 234.441,Z 594.004,A -85,B 0,C 180,E1 -20830.64,E2 -20830.64} C_VEL
LIN {X 0,Y 228.313,Z 581.815,A -85,B 0,C 180,E1 -20832.372,E2 -20832.372} C_VEL
LIN {X 0,Y 222.096,Z 570.873,A -85,B 0,C 180,E1 -20834.218,E2 -20834.218} C_VEL
LIN {X 0,Y 218.822,Z 566.275,A -85,B 0,C 180,E1 -20835.204,E2 -20835.204} C_VEL
LIN {X 0,Y 216.291,Z 562.421,A -85,B 0,C 180,E1 -20836.012,E2 -20836.012} C_VEL
LIN {X 0,Y 214.489,Z 560.131,A -85,B 0,C 180,E1 -20836.585,E2 -20836.585} C_VEL
LIN {X 0,Y 213.819,Z 557.848,A -85,B 0,C 180,E1 -20836.916,E2 -20836.916} C_VEL
LIN {X 0,Y 213.751,Z 557.858,A -85,B 0,C 180,E1 -20842.1,E2 -20842.1} C_VEL
LIN {X 0,Y 213.767,Z 557.851,A -85,B 0,C 180,E1 -20846.019,E2 -20846.019} C_VEL
LIN {X 0,Y 213.778,Z 557.85,A -85,B 0,C 180,E1 -20850.453,E2 -20850.453} C_VEL
LIN {X 0,Y 213.799,Z 557.849,A -85,B 0,C 180,E1 -20854.701,E2 -20854.701} C_VEL
LIN {X 0,Y 213.809,Z 557.845,A -85,B 0,C 180,E1 -20858.803,E2 -20858.803} C_VEL
LIN {X 0,Y 213.94,Z 557.825,A -85,B 0,C 180,E1 -20862.803,E2 -20862.803} C_VEL
LIN {X 0,Y 213.948,Z 557.823,A -85,B 0,C 180,E1 -20866.706,E2 -20866.706} C_VEL
LIN {X 0,Y 214.137,Z 557.809,A -85,B 0,C 180,E1 -20870.555,E2 -20870.555} C_VEL
LIN {X 0,Y 214.097,Z 557.813,A -85,B 0,C 180,E1 -20874.348,E2 -20874.348} C_VEL
LIN {X 0,Y 214.441,Z 557.759,A -85,B 0,C 180,E1 -20878.122,E2 -20878.122} C_VEL
LIN {X 0,Y 214.549,Z 557.758,A -85,B 0,C 180,E1 -20880,E2 -20880} C_VEL
LIN {X 0,Y 214.44,Z 557.767,A -85,B 0,C 180,E1 -20881.878,E2 -20881.878} C_VEL
LIN {X 0,Y 214.193,Z 557.796,A -85,B 0,C 180,E1 -20887.541,E2 -20887.541} C_VEL
LIN {X 0,Y 214.003,Z 557.828,A -85,B 0,C 180,E1 -20891.364,E2 -20891.364} C_VEL
LIN {X 0,Y 213.928,Z 557.834,A -85,B 0,C 180,E1 -20895.237,E2 -20895.237} C_VEL
LIN {X 0,Y 213.831,Z 557.841,A -85,B 0,C 180,E1 -20899.188,E2 -20899.188} C_VEL
LIN {X 0,Y 213.807,Z 557.842,A -85,B 0,C 180,E1 -20903.232,E2 -20903.232} C_VEL
LIN {X 0,Y 213.826,Z 557.839,A -85,B 0,C 180,E1 -20907.45,E2 -20907.45} C_VEL
LIN {X 0,Y 213.776,Z 557.856,A -85,B 0,C 180,E1 -20911.736,E2 -20911.736} C_VEL
LIN {X 0,Y 213.751,Z 557.858,A -85,B 0,C 180,E1 -20916.287,E2 -20916.287} C_VEL
LIN {X 0,Y 213.76,Z 557.859,A -85,B 0,C 180,E1 -20920.872,E2 -20920.872} C_VEL
LIN {X 0,Y 213.788,Z 557.856,A -85,B 0,C 180,E1 -20922.624,E2 -20922.624} C_VEL
LIN {X 0,Y 213.628,Z 558.913,A -85,B 0,C 180,E1 -20923.33,E2 -20923.33} C_VEL
LIN {X 0,Y 211.819,Z 563.158,A -85,B 0,C 180,E1 -20925.167,E2 -20925.167} C_VEL
LIN {X 0,Y 211.154,Z 567.81,A -85,B 0,C 180,E1 -20926.203,E2 -20926.203} C_VEL
LIN {X 0,Y 211.922,Z 571.082,A -85,B 0,C 180,E1 -20926.878,E2 -20926.878} C_VEL
LIN {X 0,Y 212.203,Z 571.586,A -85,B 0,C 180,E1 -20926.985,E2 -20926.985} C_VEL
LIN {X 0,Y 218.496,Z 582.524,A -85,B 0,C 180,E1 -20929.076,E2 -20929.076} C_VEL
LIN {X 0,Y 224.405,Z 594.001,A -85,B 0,C 180,E1 -20930.925,E2 -20930.925} C_VEL
LIN {X 0,Y 231.312,Z 609.372,A -85,B 0,C 180,E1 -20932.984,E2 -20932.984} C_VEL
LIN {X 0,Y 233.125,Z 614.594,A -85,B 0,C 180,E1 -20933.54,E2 -20933.54} C_VEL
LIN {X 0,Y 234.48,Z 624.487,A -85,B 0,C 180,E1 -20934.175,E2 -20934.175} C_VEL
LIN {X 0,Y 231.989,Z 674.719,A -85,B 0,C 180,E1 -20935.665,E2 -20935.665} C_VEL
LIN {X 0,Y 230.451,Z 688.497,A -85,B 0,C 180,E1 -20936.383,E2 -20936.383} C_VEL
LIN {X 0,Y 228.295,Z 701.468,A -85,B 0,C 180,E1 -20937.403,E2 -20937.403} C_VEL
LIN {X 0,Y 225.895,Z 712.468,A -85,B 0,C 180,E1 -20938.593,E2 -20938.593} C_VEL
LIN {X 0,Y 223.01,Z 723.964,A -85,B 0,C 180,E1 -20940.242,E2 -20940.242} C_VEL
LIN {X 0,Y 219.897,Z 734.331,A -85,B 0,C 180,E1 -20942.134,E2 -20942.134} C_VEL
LIN {X 0,Y 217.042,Z 742.814,A -85,B 0,C 180,E1 -20944.079,E2 -20944.079} C_VEL
LIN {X 0,Y 213.78,Z 752.021,A -85,B 0,C 180,E1 -20946.766,E2 -20946.766} C_VEL
LIN {X 0,Y 211.091,Z 759.433,A -85,B 0,C 180,E1 -20949.539,E2 -20949.539} C_VEL
LIN {X 0,Y 208.795,Z 765.396,A -85,B 0,C 180,E1 -20952.366,E2 -20952.366} C_VEL
LIN {X 0,Y 206.916,Z 770.117,A -85,B 0,C 180,E1 -20955.242,E2 -20955.242} C_VEL
LIN {X 0,Y 205.685,Z 773.739,A -85,B 0,C 180,E1 -20958.17,E2 -20958.17} C_VEL
LIN {X 0,Y 205.08,Z 775.616,A -85,B 0,C 180,E1 -20960.134,E2 -20960.134} C_VEL
LIN {X 0,Y 204.403,Z 778.047,A -85,B 0,C 180,E1 -20964.08,E2 -20964.08} C_VEL
LIN {X 0,Y 204.359,Z 778.922,A -85,B 0,C 180,E1 -20968.029,E2 -20968.029} C_VEL
LIN {X 0,Y 204.482,Z 778.735,A -85,B 0,C 180,E1 -20970,E2 -20970} C_VEL
LIN {X 0,Y 204.367,Z 778.14,A -85,B 0,C 180,E1 -20971.971,E2 -20971.971} C_VEL
LIN {X 0,Y 204.357,Z 777.015,A -85,B 0,C 180,E1 -20974.186,E2 -20974.186} C_VEL
LIN {X 0,Y 204.639,Z 773.912,A -85,B 0,C 180,E1 -20977.896,E2 -20977.896} C_VEL
LIN {X 0,Y 205.221,Z 770.3,A -85,B 0,C 180,E1 -20980.856,E2 -20980.856} C_VEL
LIN {X 0,Y 206.216,Z 765.57,A -85,B 0,C 180,E1 -20983.802,E2 -20983.802} C_VEL
LIN {X 0,Y 208.181,Z 758.465,A -85,B 0,C 180,E1 -20987.181,E2 -20987.181} C_VEL
LIN {X 0,Y 210.269,Z 750.915,A -85,B 0,C 180,E1 -20989.976,E2 -20989.976} C_VEL
LIN {X 0,Y 212.265,Z 742.828,A -85,B 0,C 180,E1 -20992.38,E2 -20992.38} C_VEL
LIN {X 0,Y 214.632,Z 733.164,A -85,B 0,C 180,E1 -20994.676,E2 -20994.676} C_VEL
LIN {X 0,Y 217.155,Z 722.443,A -85,B 0,C 180,E1 -20996.682,E2 -20996.682} C_VEL
LIN {X 0,Y 219.293,Z 712.067,A -85,B 0,C 180,E1 -20998.21,E2 -20998.21} C_VEL
LIN {X 0,Y 221.431,Z 699.63,A -85,B 0,C 180,E1 -20999.599,E2 -20999.599} C_VEL
LIN {X 0,Y 223.186,Z 686.518,A -85,B 0,C 180,E1 -21000.645,E2 -21000.645} C_VEL
LIN {X 0,Y 224.321,Z 673.551,A -85,B 0,C 180,E1 -21001.323,E2 -21001.323} C_VEL
LIN {X 0,Y 226.511,Z 621.313,A -85,B 0,C 180,E1 -21002.918,E2 -21002.918} C_VEL
LIN {X 0,Y 224.003,Z 601.119,A -85,B 0,C 180,E1 -21004.047,E2 -21004.047} C_VEL
LIN {X 0,Y 218.824,Z 587.953,A -85,B 0,C 180,E1 -21005.404,E2 -21005.404} C_VEL
LIN {X 0,Y 212.437,Z 573.934,A -85,B 0,C 180,E1 -21007.11,E2 -21007.11} C_VEL
LIN {X 0,Y 210.003,Z 569.195,A -85,B 0,C 180,E1 -21007.773,E2 -21007.773} C_VEL
LIN {X 0,Y 208.549,Z 565.976,A -85,B 0,C 180,E1 -21008.264,E2 -21008.264} C_VEL
LIN {X 0,Y 206.675,Z 558.739,A -85,B 0,C 180,E1 -21012.3,E2 -21012.3} C_VEL
LIN {X 0,Y 206.678,Z 558.737,A -85,B 0,C 180,E1 -21017.149,E2 -21017.149} C_VEL
LIN {X 0,Y 206.755,Z 558.732,A -85,B 0,C 180,E1 -21021.425,E2 -21021.425} C_VEL
LIN {X 0,Y 206.729,Z 558.733,A -85,B 0,C 180,E1 -21024.695,E2 -21024.695} C_VEL
LIN {X 0,Y 206.721,Z 558.735,A -85,B 0,C 180,E1 -21029.339,E2 -21029.339} C_VEL
LIN {X 0,Y 206.728,Z 558.734,A -85,B 0,C 180,E1 -21033.772,E2 -21033.772} C_VEL
LIN {X 0,Y 206.734,Z 558.729,A -85,B 0,C 180,E1 -21038.041,E2 -21038.041} C_VEL
LIN {X 0,Y 206.868,Z 558.706,A -85,B 0,C 180,E1 -21042.196,E2 -21042.196} C_VEL
LIN {X 0,Y 206.889,Z 558.712,A -85,B 0,C 180,E1 -21046.244,E2 -21046.244} C_VEL
LIN {X 0,Y 207.101,Z 558.684,A -85,B 0,C 180,E1 -21050.231,E2 -21050.231} C_VEL
LIN {X 0,Y 207.162,Z 558.679,A -85,B 0,C 180,E1 -21052.201,E2 -21052.201} C_VEL
LIN {X 0,Y 207.377,Z 558.653,A -85,B 0,C 180,E1 -21058.058,E2 -21058.058} C_VEL
LIN {X 0,Y 207.51,Z 558.634,A -85,B 0,C 180,E1 -21060,E2 -21060} C_VEL
LIN {X 0,Y 207.377,Z 558.64,A -85,B 0,C 180,E1 -21061.942,E2 -21061.942} C_VEL
LIN {X 0,Y 207.144,Z 558.677,A -85,B 0,C 180,E1 -21067.8,E2 -21067.8} C_VEL
LIN {X 0,Y 206.92,Z 558.689,A -85,B 0,C 180,E1 -21071.759,E2 -21071.759} C_VEL
LIN {X 0,Y 206.862,Z 558.717,A -85,B 0,C 180,E1 -21075.771,E2 -21075.771} C_VEL
LIN {X 0,Y 206.78,Z 558.706,A -85,B 0,C 180,E1 -21079.87,E2 -21079.87} C_VEL
LIN {X 0,Y 206.761,Z 558.73,A -85,B 0,C 180,E1 -21084.073,E2 -21084.073} C_VEL
LIN {X 0,Y 206.742,Z 558.731,A -85,B 0,C 180,E1 -21088.42,E2 -21088.42} C_VEL
LIN {X 0,Y 206.707,Z 558.735,A -85,B 0,C 180,E1 -21092.957,E2 -21092.957} C_VEL
LIN {X 0,Y 206.72,Z 558.729,A -85,B 0,C 180,E1 -21095.321,E2 -21095.321} C_VEL
LIN {X 0,Y 206.676,Z 558.739,A -85,B 0,C 180,E1 -21100.248,E2 -21100.248} C_VEL
LIN {X 0,Y 206.693,Z 558.738,A -85,B 0,C 180,E1 -21104.437,E2 -21104.437} C_VEL
LIN {X 0,Y 206.723,Z 558.732,A -85,B 0,C 180,E1 -21108.413,E2 -21108.413} C_VEL
LIN {X 0,Y 206.726,Z 558.733,A -85,B 0,C 180,E1 -21112.271,E2 -21112.271} C_VEL
LIN {X 0,Y 206.739,Z 558.732,A -85,B 0,C 180,E1 -21115.564,E2 -21115.564} C_VEL
LIN {X 0,Y 207.836,Z 561.752,A -85,B 0,C 180,E1 -21115.941,E2 -21115.941} C_VEL
LIN {X 0,Y 209.369,Z 563.925,A -85,B 0,C 180,E1 -21116.341,E2 -21116.341} C_VEL
LIN {X 0,Y 216.708,Z 576.693,A -85,B 0,C 180,E1 -21118.243,E2 -21118.243} C_VEL
LIN {X 0,Y 222.681,Z 590.078,A -85,B 0,C 180,E1 -21119.784,E2 -21119.784} C_VEL
LIN {X 0,Y 227.27,Z 602.265,A -85,B 0,C 180,E1 -21120.965,E2 -21120.965} C_VEL
LIN {X 0,Y 224.646,Z 663.433,A -85,B 0,C 180,E1 -21122.833,E2 -21122.833} C_VEL
LIN {X 0,Y 223.521,Z 676.813,A -85,B 0,C 180,E1 -21123.586,E2 -21123.586} C_VEL
LIN {X 0,Y 221.924,Z 689.83,A -85,B 0,C 180,E1 -21124.69,E2 -21124.69} C_VEL
LIN {X 0,Y 220.082,Z 700.93,A -85,B 0,C 180,E1 -21125.975,E2 -21125.975} C_VEL
LIN {X 0,Y 217.842,Z 712.448,A -85,B 0,C 180,E1 -21127.724,E2 -21127.724} C_VEL
LIN {X 0,Y 215.465,Z 722.818,A -85,B 0,C 180,E1 -21129.723,E2 -21129.723} C_VEL
LIN {X 0,Y 213.13,Z 731.312,A -85,B 0,C 180,E1 -21131.744,E2 -21131.744} C_VEL
LIN {X 0,Y 211.136,Z 739.124,A -85,B 0,C 180,E1 -21134.061,E2 -21134.061} C_VEL
LIN {X 0,Y 209.136,Z 746.868,A -85,B 0,C 180,E1 -21136.939,E2 -21136.939} C_VEL
LIN {X 0,Y 207.253,Z 753.788,A -85,B 0,C 180,E1 -21140.239,E2 -21140.239} C_VEL
LIN {X 0,Y 206.014,Z 758.473,A -85,B 0,C 180,E1 -21143.143,E2 -21143.143} C_VEL
LIN {X 0,Y 205.058,Z 762.065,A -85,B 0,C 180,E1 -21146.07,E2 -21146.07} C_VEL
LIN {X 0,Y 204.746,Z 763.918,A -85,B 0,C 180,E1 -21148.033,E2 -21148.033} C_VEL
LIN {X 0,Y 204.538,Z 765.312,A -85,B 0,C 180,E1 -21150,E2 -21150} C_VEL
LIN {X 0,Y 204.421,Z 766.307,A -85,B 0,C 180,E1 -21151.97,E2 -21151.97} C_VEL
LIN {X 0,Y 204.355,Z 766.979,A -85,B 0,C 180,E1 -21154.17,E2 -21154.17} C_VEL
LIN {X 0,Y 204.515,Z 766.964,A -85,B 0,C 180,E1 -21157.901,E2 -21157.901} C_VEL
LIN {X 0,Y 204.78,Z 766.379,A -85,B 0,C 180,E1 -21159.881,E2 -21159.881} C_VEL
LIN {X 0,Y 205.715,Z 764.039,A -85,B 0,C 180,E1 -21163.836,E2 -21163.836} C_VEL
LIN {X 0,Y 206.97,Z 761.144,A -85,B 0,C 180,E1 -21166.776,E2 -21166.776} C_VEL
LIN {X 0,Y 208.62,Z 757.209,A -85,B 0,C 180,E1 -21169.686,E2 -21169.686} C_VEL
LIN {X 0,Y 211.08,Z 751.122,A -85,B 0,C 180,E1 -21173.03,E2 -21173.03} C_VEL
LIN {X 0,Y 213.758,Z 744.453,A -85,B 0,C 180,E1 -21175.825,E2 -21175.825} C_VEL
LIN {X 0,Y 216.777,Z 736.159,A -85,B 0,C 180,E1 -21178.567,E2 -21178.567} C_VEL
LIN {X 0,Y 219.654,Z 727.604,A -85,B 0,C 180,E1 -21180.792,E2 -21180.792} C_VEL
LIN {X 0,Y 222.553,Z 718.2,A -85,B 0,C 180,E1 -21182.737,E2 -21182.737} C_VEL
LIN {X 0,Y 225.691,Z 706.506,A -85,B 0,C 180,E1 -21184.631,E2 -21184.631} C_VEL
LIN {X 0,Y 228.294,Z 694.867,A -85,B 0,C 180,E1 -21186.068,E2 -21186.068} C_VEL
LIN {X 0,Y 230.121,Z 684.027,A -85,B 0,C 180,E1 -21187.096,E2 -21187.096} C_VEL
LIN {X 0,Y 231.797,Z 670.938,A -85,B 0,C 180,E1 -21187.971,E2 -21187.971} C_VEL
LIN {X 0,Y 232.843,Z 657.876,A -85,B 0,C 180,E1 -21188.513,E2 -21188.513} C_VEL
LIN {X 0,Y 235.054,Z 610.614,A -85,B 0,C 180,E1 -21189.888,E2 -21189.888} C_VEL
LIN {X 0,Y 228.807,Z 596.228,A -85,B 0,C 180,E1 -21191.688,E2 -21191.688} C_VEL
LIN {X 0,Y 222.029,Z 582.971,A -85,B 0,C 180,E1 -21193.718,E2 -21193.718} C_VEL
LIN {X 0,Y 217.693,Z 575.549,A -85,B 0,C 180,E1 -21195.072,E2 -21195.072} C_VEL
LIN {X 0,Y 212.156,Z 567.465,A -85,B 0,C 180,E1 -21196.866,E2 -21196.866} C_VEL
LIN {X 0,Y 210.024,Z 564.188,A -85,B 0,C 180,E1 -21197.605,E2 -21197.605} C_VEL
LIN {X 0,Y 207.45,Z 561.08,A -85,B 0,C 180,E1 -21198.491,E2 -21198.491} C_VEL
LIN {X 0,Y 206.723,Z 558.714,A -85,B 0,C 180,E1 -21198.874,E2 -21198.874} C_VEL
LIN {X 0,Y 206.699,Z 558.735,A -85,B 0,C 180,E1 -21202.264,E2 -21202.264} C_VEL
LIN {X 0,Y 206.73,Z 558.735,A -85,B 0,C 180,E1 -21204.694,E2 -21204.694} C_VEL
LIN {X 0,Y 206.721,Z 558.727,A -85,B 0,C 180,E1 -21209.338,E2 -21209.338} C_VEL
LIN {X 0,Y 206.729,Z 558.724,A -85,B 0,C 180,E1 -21213.771,E2 -21213.771} C_VEL
LIN {X 0,Y 206.754,Z 558.72,A -85,B 0,C 180,E1 -21218.042,E2 -21218.042} C_VEL
LIN {X 0,Y 206.87,Z 558.705,A -85,B 0,C 180,E1 -21222.196,E2 -21222.196} C_VEL
LIN {X 0,Y 206.891,Z 558.704,A -85,B 0,C 180,E1 -21226.244,E2 -21226.244} C_VEL
LIN {X 0,Y 207.096,Z 558.689,A -85,B 0,C 180,E1 -21230.23,E2 -21230.23} C_VEL
LIN {X 0,Y 207.058,Z 558.689,A -85,B 0,C 180,E1 -21234.155,E2 -21234.155} C_VEL
LIN {X 0,Y 207.378,Z 558.638,A -85,B 0,C 180,E1 -21238.058,E2 -21238.058} C_VEL
LIN {X 0,Y 207.514,Z 558.635,A -85,B 0,C 180,E1 -21240,E2 -21240} C_VEL
LIN {X 0,Y 207.377,Z 558.645,A -85,B 0,C 180,E1 -21241.942,E2 -21241.942} C_VEL
LIN {X 0,Y 207.136,Z 558.672,A -85,B 0,C 180,E1 -21247.8,E2 -21247.8} C_VEL
LIN {X 0,Y 206.926,Z 558.709,A -85,B 0,C 180,E1 -21251.758,E2 -21251.758} C_VEL
LIN {X 0,Y 206.862,Z 558.717,A -85,B 0,C 180,E1 -21255.771,E2 -21255.771} C_VEL
LIN {X 0,Y 206.774,Z 558.725,A -85,B 0,C 180,E1 -21259.87,E2 -21259.87} C_VEL
LIN {X 0,Y 206.743,Z 558.726,A -85,B 0,C 180,E1 -21264.074,E2 -21264.074} C_VEL
LIN {X 0,Y 206.741,Z 558.726,A -85,B 0,C 180,E1 -21268.419,E2 -21268.419} C_VEL
LIN {X 0,Y 206.706,Z 558.737,A -85,B 0,C 180,E1 -21272.956,E2 -21272.956} C_VEL
LIN {X 0,Y 206.722,Z 558.734,A -85,B 0,C 180,E1 -21277.731,E2 -21277.731} C_VEL
LIN {X 0,Y 206.71,Z 558.751,A -85,B 0,C 180,E1 -21281.184,E2 -21281.184} C_VEL
LIN {X 0,Y 208.595,Z 565.493,A -85,B 0,C 180,E1 -21285.678,E2 -21285.678} C_VEL
LIN {X 0,Y 210.947,Z 569.712,A -85,B 0,C 180,E1 -21286.557,E2 -21286.557} C_VEL
LIN {X 0,Y 212.203,Z 571.586,A -85,B 0,C 180,E1 -21286.985,E2 -21286.985} C_VEL
LIN {X 0,Y 213.727,Z 574.601,A -85,B 0,C 180,E1 -21287.526,E2 -21287.526} C_VEL
LIN {X 0,Y 215.375,Z 579.736,A -85,B 0,C 180,E1 -21288.182,E2 -21288.182} C_VEL
LIN {X 0,Y 218.072,Z 592.669,A -85,B 0,C 180,E1 -21289.417,E2 -21289.417} C_VEL
LIN {X 0,Y 219.691,Z 597.947,A -85,B 0,C 180,E1 -21290.026,E2 -21290.026} C_VEL
LIN {X 0,Y 220.404,Z 599.581,A -85,B 0,C 180,E1 -21290.261,E2 -21290.261} C_VEL
LIN {X 0,Y 226.358,Z 613.168,A -85,B 0,C 180,E1 -21292.127,E2 -21292.127} C_VEL
LIN {X 0,Y 227.697,Z 616.795,A -85,B 0,C 180,E1 -21292.549,E2 -21292.549} C_VEL
LIN {X 0,Y 228.84,Z 626.023,A -85,B 0,C 180,E1 -21293.145,E2 -21293.145} C_VEL
LIN {X 0,Y 226.261,Z 674.984,A -85,B 0,C 180,E1 -21294.626,E2 -21294.626} C_VEL
LIN {X 0,Y 224.677,Z 688.499,A -85,B 0,C 180,E1 -21295.346,E2 -21295.346} C_VEL
LIN {X 0,Y 222.588,Z 700.761,A -85,B 0,C 180,E1 -21296.323,E2 -21296.323} C_VEL
LIN {X 0,Y 219.886,Z 712.674,A -85,B 0,C 180,E1 -21297.632,E2 -21297.632} C_VEL
LIN {X 0,Y 216.88,Z 724.095,A -85,B 0,C 180,E1 -21299.312,E2 -21299.312} C_VEL
LIN {X 0,Y 213.641,Z 734.404,A -85,B 0,C 180,E1 -21301.243,E2 -21301.243} C_VEL
LIN {X 0,Y 210.68,Z 742.839,A -85,B 0,C 180,E1 -21303.235,E2 -21303.235} C_VEL
LIN {X 0,Y 207.257,Z 751.992,A -85,B 0,C 180,E1 -21305.989,E2 -21305.989} C_VEL
LIN {X 0,Y 204.455,Z 759.373,A -85,B 0,C 180,E1 -21308.843,E2 -21308.843} C_VEL
LIN {X 0,Y 202.037,Z 765.309,A -85,B 0,C 180,E1 -21311.756,E2 -21311.756} C_VEL
LIN {X 0,Y 200.041,Z 770.004,A -85,B 0,C 180,E1 -21314.723,E2 -21314.723} C_VEL
LIN {X 0,Y 198.7,Z 773.602,A -85,B 0,C 180,E1 -21317.748,E2 -21317.748} C_VEL
LIN {X 0,Y 198.054,Z 775.462,A -85,B 0,C 180,E1 -21319.78,E2 -21319.78} C_VEL
LIN {X 0,Y 197.342,Z 777.869,A -85,B 0,C 180,E1 -21323.867,E2 -21323.867} C_VEL
LIN {X 0,Y 197.193,Z 778.577,A -85,B 0,C 180,E1 -21326.309,E2 -21326.309} C_VEL
LIN {X 0,Y 197.381,Z 778.515,A -85,B 0,C 180,E1 -21330,E2 -21330} C_VEL
LIN {X 0,Y 197.248,Z 776.998,A -85,B 0,C 180,E1 -21333.931,E2 -21333.931} C_VEL
LIN {X 0,Y 197.342,Z 775.51,A -85,B 0,C 180,E1 -21336.133,E2 -21336.133} C_VEL
LIN {X 0,Y 197.775,Z 772.561,A -85,B 0,C 180,E1 -21339.201,E2 -21339.201} C_VEL
LIN {X 0,Y 198.54,Z 768.563,A -85,B 0,C 180,E1 -21342.262,E2 -21342.262} C_VEL
LIN {X 0,Y 200.091,Z 762.41,A -85,B 0,C 180,E1 -21345.795,E2 -21345.795} C_VEL
LIN {X 0,Y 201.989,Z 755.691,A -85,B 0,C 180,E1 -21348.774,E2 -21348.774} C_VEL
LIN {X 0,Y 204.237,Z 747.932,A -85,B 0,C 180,E1 -21351.505,E2 -21351.505} C_VEL
LIN {X 0,Y 206.593,Z 738.765,A -85,B 0,C 180,E1 -21354.093,E2 -21354.093} C_VEL
LIN {X 0,Y 209.355,Z 728.173,A -85,B 0,C 180,E1 -21356.41,E2 -21356.41} C_VEL
LIN {X 0,Y 211.77,Z 717.672,A -85,B 0,C 180,E1 -21358.223,E2 -21358.223} C_VEL
LIN {X 0,Y 214.05,Z 706.096,A -85,B 0,C 180,E1 -21359.775,E2 -21359.775} C_VEL
LIN {X 0,Y 216.002,Z 694.069,A -85,B 0,C 180,E1 -21360.962,E2 -21360.962} C_VEL
LIN {X 0,Y 217.603,Z 680.851,A -85,B 0,C 180,E1 -21361.874,E2 -21361.874} C_VEL
LIN {X 0,Y 218.474,Z 667.922,A -85,B 0,C 180,E1 -21362.43,E2 -21362.43} C_VEL
LIN {X 0,Y 220.374,Z 621.375,A -85,B 0,C 180,E1 -21363.874,E2 -21363.874} C_VEL
LIN {X 0,Y 218.122,Z 603.311,A -85,B 0,C 180,E1 -21364.934,E2 -21364.934} C_VEL
LIN {X 0,Y 212.369,Z 588.831,A -85,B 0,C 180,E1 -21366.522,E2 -21366.522} C_VEL
LIN {X 0,Y 205.656,Z 574.352,A -85,B 0,C 180,E1 -21368.428,E2 -21368.428} C_VEL
LIN {X 0,Y 201.232,Z 565.775,A -85,B 0,C 180,E1 -21369.794,E2 -21369.794} C_VEL
LIN {X 0,Y 199.601,Z 559.618,A -85,B 0,C 180,E1 -21373.477,E2 -21373.477} C_VEL
LIN {X 0,Y 199.632,Z 559.619,A -85,B 0,C 180,E1 -21378.018,E2 -21378.018} C_VEL
LIN {X 0,Y 199.675,Z 559.611,A -85,B 0,C 180,E1 -21380.743,E2 -21380.743} C_VEL
LIN {X 0,Y 199.632,Z 559.617,A -85,B 0,C 180,E1 -21385.717,E2 -21385.717} C_VEL
LIN {X 0,Y 199.701,Z 559.605,A -85,B 0,C 180,E1 -21388.137,E2 -21388.137} C_VEL
LIN {X 0,Y 199.683,Z 559.605,A -85,B 0,C 180,E1 -21392.771,E2 -21392.771} C_VEL
LIN {X 0,Y 199.71,Z 559.599,A -85,B 0,C 180,E1 -21397.226,E2 -21397.226} C_VEL
LIN {X 0,Y 199.792,Z 559.589,A -85,B 0,C 180,E1 -21401.758,E2 -21401.758} C_VEL
LIN {X 0,Y 199.829,Z 559.593,A -85,B 0,C 180,E1 -21405.748,E2 -21405.748} C_VEL
LIN {X 0,Y 200.067,Z 559.556,A -85,B 0,C 180,E1 -21409.884,E2 -21409.884} C_VEL
LIN {X 0,Y 200.029,Z 559.561,A -85,B 0,C 180,E1 -21413.95,E2 -21413.95} C_VEL
LIN {X 0,Y 200.317,Z 559.532,A -85,B 0,C 180,E1 -21417.99,E2 -21417.99} C_VEL
LIN {X 0,Y 200.474,Z 559.51,A -85,B 0,C 180,E1 -21420,E2 -21420} C_VEL
LIN {X 0,Y 200.025,Z 559.562,A -85,B 0,C 180,E1 -21424.03,E2 -21424.03} C_VEL
LIN {X 0,Y 200.091,Z 559.554,A -85,B 0,C 180,E1 -21428.077,E2 -21428.077} C_VEL
LIN {X 0,Y 199.87,Z 559.57,A -85,B 0,C 180,E1 -21432.18,E2 -21432.18} C_VEL
LIN {X 0,Y 199.8,Z 559.595,A -85,B 0,C 180,E1 -21436.344,E2 -21436.344} C_VEL
LIN {X 0,Y 199.697,Z 559.589,A -85,B 0,C 180,E1 -21440.606,E2 -21440.606} C_VEL
LIN {X 0,Y 199.67,Z 559.614,A -85,B 0,C 180,E1 -21444.985,E2 -21444.985} C_VEL
LIN {X 0,Y 199.673,Z 559.613,A -85,B 0,C 180,E1 -21449.523,E2 -21449.523} C_VEL
LIN {X 0,Y 199.662,Z 559.611,A -85,B 0,C 180,E1 -21452.353,E2 -21452.353} C_VEL
LIN {X 0,Y 199.617,Z 559.601,A -85,B 0,C 180,E1 -21456.765,E2 -21456.765} C_VEL
LIN {X 0,Y 199.639,Z 559.605,A -85,B 0,C 180,E1 -21459.321,E2 -21459.321} C_VEL
LIN {X 0,Y 199.618,Z 559.617,A -85,B 0,C 180,E1 -21462.325,E2 -21462.325} C_VEL
LIN {X 0,Y 199.651,Z 559.614,A -85,B 0,C 180,E1 -21465.25,E2 -21465.25} C_VEL
LIN {X 0,Y 199.666,Z 559.611,A -85,B 0,C 180,E1 -21468.028,E2 -21468.028} C_VEL
LIN {X 0,Y 199.68,Z 559.61,A -85,B 0,C 180,E1 -21470.744,E2 -21470.744} C_VEL
LIN {X 0,Y 199.67,Z 559.702,A -85,B 0,C 180,E1 -21474.1,E2 -21474.1} C_VEL
LIN {X 0,Y 200.743,Z 562.572,A -85,B 0,C 180,E1 -21474.469,E2 -21474.469} C_VEL
LIN {X 0,Y 202.423,Z 564.91,A -85,B 0,C 180,E1 -21474.94,E2 -21474.94} C_VEL
LIN {X 0,Y 210.503,Z 578.578,A -85,B 0,C 180,E1 -21477.167,E2 -21477.167} C_VEL
LIN {X 0,Y 215.495,Z 589.228,A -85,B 0,C 180,E1 -21478.519,E2 -21478.519} C_VEL
LIN {X 0,Y 221.1,Z 603.778,A -85,B 0,C 180,E1 -21480.039,E2 -21480.039} C_VEL
LIN {X 0,Y 219.351,Z 646.436,A -85,B 0,C 180,E1 -21481.36,E2 -21481.36} C_VEL
LIN {X 0,Y 218.367,Z 665.934,A -85,B 0,C 180,E1 -21482.037,E2 -21482.037} C_VEL
LIN {X 0,Y 217.135,Z 678.655,A -85,B 0,C 180,E1 -21482.806,E2 -21482.806} C_VEL
LIN {X 0,Y 215.564,Z 690.677,A -85,B 0,C 180,E1 -21483.888,E2 -21483.888} C_VEL
LIN {X 0,Y 213.633,Z 701.624,A -85,B 0,C 180,E1 -21485.201,E2 -21485.201} C_VEL
LIN {X 0,Y 211.319,Z 713.05,A -85,B 0,C 180,E1 -21486.998,E2 -21486.998} C_VEL
LIN {X 0,Y 208.854,Z 723.352,A -85,B 0,C 180,E1 -21489.052,E2 -21489.052} C_VEL
LIN {X 0,Y 206.429,Z 731.79,A -85,B 0,C 180,E1 -21491.13,E2 -21491.13} C_VEL
LIN {X 0,Y 204.345,Z 739.552,A -85,B 0,C 180,E1 -21493.517,E2 -21493.517} C_VEL
LIN {X 0,Y 202.236,Z 747.245,A -85,B 0,C 180,E1 -21496.485,E2 -21496.485} C_VEL
LIN {X 0,Y 200.287,Z 754.131,A -85,B 0,C 180,E1 -21499.895,E2 -21499.895} C_VEL
LIN {X 0,Y 198.985,Z 758.787,A -85,B 0,C 180,E1 -21502.899,E2 -21502.899} C_VEL
LIN {X 0,Y 197.994,Z 762.352,A -85,B 0,C 180,E1 -21505.929,E2 -21505.929} C_VEL
LIN {X 0,Y 197.667,Z 764.185,A -85,B 0,C 180,E1 -21507.962,E2 -21507.962} C_VEL
LIN {X 0,Y 197.455,Z 765.559,A -85,B 0,C 180,E1 -21510,E2 -21510} C_VEL
LIN {X 0,Y 197.324,Z 766.543,A -85,B 0,C 180,E1 -21512.041,E2 -21512.041} C_VEL
LIN {X 0,Y 197.287,Z 767.146,A -85,B 0,C 180,E1 -21514.085,E2 -21514.085} C_VEL
LIN {X 0,Y 197.299,Z 767.363,A -85,B 0,C 180,E1 -21516.134,E2 -21516.134} C_VEL
LIN {X 0,Y 197.452,Z 767.151,A -85,B 0,C 180,E1 -21518.185,E2 -21518.185} C_VEL
LIN {X 0,Y 198.168,Z 765.57,A -85,B 0,C 180,E1 -21522.286,E2 -21522.286} C_VEL
LIN {X 0,Y 198.78,Z 764.182,A -85,B 0,C 180,E1 -21524.329,E2 -21524.329} C_VEL
LIN {X 0,Y 200.114,Z 761.265,A -85,B 0,C 180,E1 -21527.368,E2 -21527.368} C_VEL
LIN {X 0,Y 201.881,Z 757.301,A -85,B 0,C 180,E1 -21530.372,E2 -21530.372} C_VEL
LIN {X 0,Y 204.509,Z 751.171,A -85,B 0,C 180,E1 -21533.815,E2 -21533.815} C_VEL
LIN {X 0,Y 207.329,Z 744.467,A -85,B 0,C 180,E1 -21536.688,E2 -21536.688} C_VEL
LIN {X 0,Y 210.487,Z 736.164,A -85,B 0,C 180,E1 -21539.49,E2 -21539.49} C_VEL
LIN {X 0,Y 213.541,Z 727.505,A -85,B 0,C 180,E1 -21541.774,E2 -21541.774} C_VEL
LIN {X 0,Y 216.895,Z 716.86,A -85,B 0,C 180,E1 -21543.982,E2 -21543.982} C_VEL
LIN {X 0,Y 219.868,Z 706.267,A -85,B 0,C 180,E1 -21545.686,E2 -21545.686} C_VEL
LIN {X 0,Y 222.549,Z 694.452,A -85,B 0,C 180,E1 -21547.153,E2 -21547.153} C_VEL
LIN {X 0,Y 224.462,Z 683.42,A -85,B 0,C 180,E1 -21548.197,E2 -21548.197} C_VEL
LIN {X 0,Y 226.171,Z 670.235,A -85,B 0,C 180,E1 -21549.074,E2 -21549.074} C_VEL
LIN {X 0,Y 227.206,Z 657.262,A -85,B 0,C 180,E1 -21549.598,E2 -21549.598} C_VEL
LIN {X 0,Y 229.34,Z 612.531,A -85,B 0,C 180,E1 -21550.932,E2 -21550.932} C_VEL
LIN {X 0,Y 223.245,Z 598.618,A -85,B 0,C 180,E1 -21552.785,E2 -21552.785} C_VEL
LIN {X 0,Y 217.204,Z 586.755,A -85,B 0,C 180,E1 -21554.697,E2 -21554.697} C_VEL
LIN {X 0,Y 213.036,Z 579.661,A -85,B 0,C 180,E1 -21556.066,E2 -21556.066} C_VEL
LIN {X 0,Y 208.054,Z 572.395,A -85,B 0,C 180,E1 -21557.764,E2 -21557.764} C_VEL
LIN {X 0,Y 205.685,Z 568.896,A -85,B 0,C 180,E1 -21558.621,E2 -21558.621} C_VEL
LIN {X 0,Y 203.476,Z 565.843,A -85,B 0,C 180,E1 -21559.44,E2 -21559.44} C_VEL
LIN {X 0,Y 202.57,Z 564.5,A -85,B 0,C 180,E1 -21559.79,E2 -21559.79} C_VEL
LIN {X 0,Y 200.532,Z 562.238,A -85,B 0,C 180,E1 -21560.557,E2 -21560.557} C_VEL
LIN {X 0,Y 199.672,Z 559.607,A -85,B 0,C 180,E1 -21561.023,E2 -21561.023} C_VEL
LIN {X 0,Y 199.632,Z 559.612,A -85,B 0,C 180,E1 -21565.717,E2 -21565.717} C_VEL
LIN {X 0,Y 199.702,Z 559.61,A -85,B 0,C 180,E1 -21568.137,E2 -21568.137} C_VEL
LIN {X 0,Y 199.684,Z 559.604,A -85,B 0,C 180,E1 -21572.771,E2 -21572.771} C_VEL
LIN {X 0,Y 199.735,Z 559.595,A -85,B 0,C 180,E1 -21577.228,E2 -21577.228} C_VEL
LIN {X 0,Y 199.793,Z 559.587,A -85,B 0,C 180,E1 -21581.757,E2 -21581.757} C_VEL
LIN {X 0,Y 199.832,Z 559.588,A -85,B 0,C 180,E1 -21585.748,E2 -21585.748} C_VEL
LIN {X 0,Y 200.019,Z 559.57,A -85,B 0,C 180,E1 -21589.881,E2 -21589.881} C_VEL
LIN {X 0,Y 200.019,Z 559.564,A -85,B 0,C 180,E1 -21593.949,E2 -21593.949} C_VEL
LIN {X 0,Y 200.317,Z 559.517,A -85,B 0,C 180,E1 -21597.989,E2 -21597.989} C_VEL
LIN {X 0,Y 200.478,Z 559.511,A -85,B 0,C 180,E1 -21600,E2 -21600} C_VEL
LIN {X 0,Y 200.022,Z 559.557,A -85,B 0,C 180,E1 -21604.029,E2 -21604.029} C_VEL
LIN {X 0,Y 200.084,Z 559.549,A -85,B 0,C 180,E1 -21608.077,E2 -21608.077} C_VEL
LIN {X 0,Y 199.874,Z 559.582,A -85,B 0,C 180,E1 -21612.179,E2 -21612.179} C_VEL
LIN {X 0,Y 199.8,Z 559.598,A -85,B 0,C 180,E1 -21616.344,E2 -21616.344} C_VEL
LIN {X 0,Y 199.686,Z 559.612,A -85,B 0,C 180,E1 -21620.607,E2 -21620.607} C_VEL
LIN {X 0,Y 199.661,Z 559.615,A -85,B 0,C 180,E1 -21624.986,E2 -21624.986} C_VEL
LIN {X 0,Y 199.672,Z 559.613,A -85,B 0,C 180,E1 -21629.523,E2 -21629.523} C_VEL
LIN {X 0,Y 199.661,Z 559.612,A -85,B 0,C 180,E1 -21632.353,E2 -21632.353} C_VEL
LIN {X 0,Y 199.65,Z 559.617,A -85,B 0,C 180,E1 -21636.757,E2 -21636.757} C_VEL
LIN {X 0,Y 199.671,Z 559.696,A -85,B 0,C 180,E1 -21639.477,E2 -21639.477} C_VEL
LIN {X 0,Y 201.286,Z 565.346,A -85,B 0,C 180,E1 -21643.494,E2 -21643.494} C_VEL
LIN {X 0,Y 203.719,Z 569.516,A -85,B 0,C 180,E1 -21644.467,E2 -21644.467} C_VEL
LIN {X 0,Y 205.175,Z 571.702,A -85,B 0,C 180,E1 -21645.014,E2 -21645.014} C_VEL
LIN {X 0,Y 208.938,Z 577.961,A -85,B 0,C 180,E1 -21646.398,E2 -21646.398} C_VEL
LIN {X 0,Y 213.882,Z 586.587,A -85,B 0,C 180,E1 -21648.113,E2 -21648.113} C_VEL
LIN {X 0,Y 219.615,Z 597.806,A -85,B 0,C 180,E1 -21650.003,E2 -21650.003} C_VEL
LIN {X 0,Y 220.404,Z 599.581,A -85,B 0,C 180,E1 -21650.261,E2 -21650.261} C_VEL
LIN {X 0,Y 221.531,Z 603.022,A -85,B 0,C 180,E1 -21650.662,E2 -21650.662} C_VEL
LIN {X 0,Y 222.157,Z 609.429,A -85,B 0,C 180,E1 -21651.07,E2 -21651.07} C_VEL
LIN {X 0,Y 222.442,Z 620.163,A -85,B 0,C 180,E1 -21651.579,E2 -21651.579} C_VEL
LIN {X 0,Y 223.239,Z 627.5,A -85,B 0,C 180,E1 -21652.052,E2 -21652.052} C_VEL
LIN {X 0,Y 220.683,Z 674.327,A -85,B 0,C 180,E1 -21653.488,E2 -21653.488} C_VEL
LIN {X 0,Y 219.112,Z 687.891,A -85,B 0,C 180,E1 -21654.222,E2 -21654.222} C_VEL
LIN {X 0,Y 216.972,Z 700.025,A -85,B 0,C 180,E1 -21655.188,E2 -21655.188} C_VEL
LIN {X 0,Y 214.346,Z 711.299,A -85,B 0,C 180,E1 -21656.407,E2 -21656.407} C_VEL
LIN {X 0,Y 211.199,Z 722.936,A -85,B 0,C 180,E1 -21658.112,E2 -21658.112} C_VEL
LIN {X 0,Y 207.781,Z 733.409,A -85,B 0,C 180,E1 -21660.073,E2 -21660.073} C_VEL
LIN {X 0,Y 204.352,Z 742.857,A -85,B 0,C 180,E1 -21662.337,E2 -21662.337} C_VEL
LIN {X 0,Y 200.76,Z 751.963,A -85,B 0,C 180,E1 -21665.161,E2 -21665.161} C_VEL
LIN {X 0,Y 197.851,Z 759.314,A -85,B 0,C 180,E1 -21668.101,E2 -21668.101} C_VEL
LIN {X 0,Y 195.286,Z 765.221,A -85,B 0,C 180,E1 -21671.102,E2 -21671.102} C_VEL
LIN {X 0,Y 193.163,Z 769.891,A -85,B 0,C 180,E1 -21674.165,E2 -21674.165} C_VEL
LIN {X 0,Y 191.738,Z 773.466,A -85,B 0,C 180,E1 -21677.296,E2 -21677.296} C_VEL
LIN {X 0,Y 191.047,Z 775.307,A -85,B 0,C 180,E1 -21679.401,E2 -21679.401} C_VEL
LIN {X 0,Y 190.279,Z 777.69,A -85,B 0,C 180,E1 -21683.638,E2 -21683.638} C_VEL
LIN {X 0,Y 190.11,Z 778.41,A -85,B 0,C 180,E1 -21686.504,E2 -21686.504} C_VEL
LIN {X 0,Y 190.283,Z 778.295,A -85,B 0,C 180,E1 -21690,E2 -21690} C_VEL
LIN {X 0,Y 190.16,Z 776.939,A -85,B 0,C 180,E1 -21693.736,E2 -21693.736} C_VEL
LIN {X 0,Y 190.279,Z 775.252,A -85,B 0,C 180,E1 -21696.362,E2 -21696.362} C_VEL
LIN {X 0,Y 190.733,Z 772.283,A -85,B 0,C 180,E1 -21699.544,E2 -21699.544} C_VEL
LIN {X 0,Y 191.582,Z 768.262,A -85,B 0,C 180,E1 -21702.715,E2 -21702.715} C_VEL
LIN {X 0,Y 193.242,Z 762.073,A -85,B 0,C 180,E1 -21706.371,E2 -21706.371} C_VEL
LIN {X 0,Y 195.244,Z 755.324,A -85,B 0,C 180,E1 -21709.448,E2 -21709.448} C_VEL
LIN {X 0,Y 197.412,Z 748.216,A -85,B 0,C 180,E1 -21712.036,E2 -21712.036} C_VEL
LIN {X 0,Y 199.59,Z 740.153,A -85,B 0,C 180,E1 -21714.44,E2 -21714.44} C_VEL
LIN {X 0,Y 202.387,Z 730.02,A -85,B 0,C 180,E1 -21716.835,E2 -21716.835} C_VEL
LIN {X 0,Y 204.857,Z 719.96,A -85,B 0,C 180,E1 -21718.704,E2 -21718.704} C_VEL
LIN {X 0,Y 207.149,Z 709.005,A -85,B 0,C 180,E1 -21720.309,E2 -21720.309} C_VEL
LIN {X 0,Y 209.365,Z 696.906,A -85,B 0,C 180,E1 -21721.634,E2 -21721.634} C_VEL
LIN {X 0,Y 211.069,Z 684.398,A -85,B 0,C 180,E1 -21722.619,E2 -21722.619} C_VEL
LIN {X 0,Y 212.214,Z 671.191,A -85,B 0,C 180,E1 -21723.278,E2 -21723.278} C_VEL
LIN {X 0,Y 214.382,Z 622.979,A -85,B 0,C 180,E1 -21724.811,E2 -21724.811} C_VEL
LIN {X 0,Y 212.391,Z 605.896,A -85,B 0,C 180,E1 -21725.835,E2 -21725.835} C_VEL
LIN {X 0,Y 206.864,Z 591.867,A -85,B 0,C 180,E1 -21727.448,E2 -21727.448} C_VEL
LIN {X 0,Y 200.67,Z 578.384,A -85,B 0,C 180,E1 -21729.305,E2 -21729.305} C_VEL
LIN {X 0,Y 195.671,Z 569.152,A -85,B 0,C 180,E1 -21730.85,E2 -21730.85} C_VEL
LIN {X 0,Y 193.842,Z 565.502,A -85,B 0,C 180,E1 -21731.52,E2 -21731.52} C_VEL
LIN {X 0,Y 192.558,Z 560.497,A -85,B 0,C 180,E1 -21734.718,E2 -21734.718} C_VEL
LIN {X 0,Y 192.577,Z 560.492,A -85,B 0,C 180,E1 -21740.029,E2 -21740.029} C_VEL
LIN {X 0,Y 192.599,Z 560.491,A -85,B 0,C 180,E1 -21744.279,E2 -21744.279} C_VEL
LIN {X 0,Y 192.605,Z 560.493,A -85,B 0,C 180,E1 -21749.28,E2 -21749.28} C_VEL
LIN {X 0,Y 192.661,Z 560.477,A -85,B 0,C 180,E1 -21751.692,E2 -21751.692} C_VEL
LIN {X 0,Y 192.681,Z 560.475,A -85,B 0,C 180,E1 -21756.346,E2 -21756.346} C_VEL
LIN {X 0,Y 192.728,Z 560.47,A -85,B 0,C 180,E1 -21761.458,E2 -21761.458} C_VEL
LIN {X 0,Y 192.758,Z 560.474,A -85,B 0,C 180,E1 -21765.213,E2 -21765.213} C_VEL
LIN {X 0,Y 192.978,Z 560.436,A -85,B 0,C 180,E1 -21769.508,E2 -21769.508} C_VEL
LIN {X 0,Y 193.057,Z 560.438,A -85,B 0,C 180,E1 -21771.627,E2 -21771.627} C_VEL
LIN {X 0,Y 193.259,Z 560.411,A -85,B 0,C 180,E1 -21777.916,E2 -21777.916} C_VEL
LIN {X 0,Y 193.438,Z 560.387,A -85,B 0,C 180,E1 -21780,E2 -21780} C_VEL
LIN {X 0,Y 192.971,Z 560.441,A -85,B 0,C 180,E1 -21784.177,E2 -21784.177} C_VEL
LIN {X 0,Y 193.037,Z 560.432,A -85,B 0,C 180,E1 -21788.374,E2 -21788.374} C_VEL
LIN {X 0,Y 192.798,Z 560.454,A -85,B 0,C 180,E1 -21792.634,E2 -21792.634} C_VEL
LIN {X 0,Y 192.754,Z 560.471,A -85,B 0,C 180,E1 -21796.959,E2 -21796.959} C_VEL
LIN {X 0,Y 192.633,Z 560.473,A -85,B 0,C 180,E1 -21801.398,E2 -21801.398} C_VEL
LIN {X 0,Y 192.662,Z 560.486,A -85,B 0,C 180,E1 -21804.225,E2 -21804.225} C_VEL
LIN {X 0,Y 192.648,Z 560.487,A -85,B 0,C 180,E1 -21808.893,E2 -21808.893} C_VEL
LIN {X 0,Y 192.599,Z 560.493,A -85,B 0,C 180,E1 -21813.186,E2 -21813.186} C_VEL
LIN {X 0,Y 192.595,Z 560.476,A -85,B 0,C 180,E1 -21816.603,E2 -21816.603} C_VEL
LIN {X 0,Y 192.546,Z 560.501,A -85,B 0,C 180,E1 -21821.073,E2 -21821.073} C_VEL
LIN {X 0,Y 192.596,Z 560.49,A -85,B 0,C 180,E1 -21826.107,E2 -21826.107} C_VEL
LIN {X 0,Y 192.591,Z 560.494,A -85,B 0,C 180,E1 -21830.026,E2 -21830.026} C_VEL
LIN {X 0,Y 192.586,Z 560.495,A -85,B 0,C 180,E1 -21832.432,E2 -21832.432} C_VEL
LIN {X 0,Y 193.656,Z 563.443,A -85,B 0,C 180,E1 -21832.858,E2 -21832.858} C_VEL
LIN {X 0,Y 195.351,Z 565.625,A -85,B 0,C 180,E1 -21833.369,E2 -21833.369} C_VEL
LIN {X 0,Y 203.884,Z 579.721,A -85,B 0,C 180,E1 -21835.893,E2 -21835.893} C_VEL
LIN {X 0,Y 208.058,Z 587.884,A -85,B 0,C 180,E1 -21837.077,E2 -21837.077} C_VEL
LIN {X 0,Y 213.924,Z 602.418,A -85,B 0,C 180,E1 -21838.759,E2 -21838.759} C_VEL
LIN {X 0,Y 215.158,Z 606.366,A -85,B 0,C 180,E1 -21839.132,E2 -21839.132} C_VEL
LIN {X 0,Y 212.405,Z 664.108,A -85,B 0,C 180,E1 -21840.974,E2 -21840.974} C_VEL
LIN {X 0,Y 211.215,Z 676.848,A -85,B 0,C 180,E1 -21841.714,E2 -21841.714} C_VEL
LIN {X 0,Y 209.559,Z 689.395,A -85,B 0,C 180,E1 -21842.811,E2 -21842.811} C_VEL
LIN {X 0,Y 207.518,Z 700.736,A -85,B 0,C 180,E1 -21844.149,E2 -21844.149} C_VEL
LIN {X 0,Y 205.119,Z 712.37,A -85,B 0,C 180,E1 -21845.992,E2 -21845.992} C_VEL
LIN {X 0,Y 202.533,Z 722.823,A -85,B 0,C 180,E1 -21848.098,E2 -21848.098} C_VEL
LIN {X 0,Y 199.76,Z 732.263,A -85,B 0,C 180,E1 -21850.475,E2 -21850.475} C_VEL
LIN {X 0,Y 197.582,Z 739.974,A -85,B 0,C 180,E1 -21852.936,E2 -21852.936} C_VEL
LIN {X 0,Y 195.399,Z 747.51,A -85,B 0,C 180,E1 -21855.95,E2 -21855.95} C_VEL
LIN {X 0,Y 193.328,Z 754.474,A -85,B 0,C 180,E1 -21859.528,E2 -21859.528} C_VEL
LIN {X 0,Y 191.961,Z 759.101,A -85,B 0,C 180,E1 -21862.638,E2 -21862.638} C_VEL
LIN {X 0,Y 190.934,Z 762.638,A -85,B 0,C 180,E1 -21865.778,E2 -21865.778} C_VEL
LIN {X 0,Y 190.591,Z 764.448,A -85,B 0,C 180,E1 -21867.887,E2 -21867.887} C_VEL
LIN {X 0,Y 190.354,Z 765.807,A -85,B 0,C 180,E1 -21870,E2 -21870} C_VEL
LIN {X 0,Y 190.194,Z 767.288,A -85,B 0,C 180,E1 -21873.88,E2 -21873.88} C_VEL
LIN {X 0,Y 190.215,Z 767.566,A -85,B 0,C 180,E1 -21876.364,E2 -21876.364} C_VEL
LIN {X 0,Y 190.407,Z 767.338,A -85,B 0,C 180,E1 -21878.49,E2 -21878.49} C_VEL
LIN {X 0,Y 191.172,Z 765.733,A -85,B 0,C 180,E1 -21882.743,E2 -21882.743} C_VEL
LIN {X 0,Y 191.867,Z 764.321,A -85,B 0,C 180,E1 -21884.857,E2 -21884.857} C_VEL
LIN {X 0,Y 193.288,Z 761.381,A -85,B 0,C 180,E1 -21888.002,E2 -21888.002} C_VEL
LIN {X 0,Y 195.182,Z 757.39,A -85,B 0,C 180,E1 -21891.104,E2 -21891.104} C_VEL
LIN {X 0,Y 197.974,Z 751.22,A -85,B 0,C 180,E1 -21894.652,E2 -21894.652} C_VEL
LIN {X 0,Y 200.968,Z 744.481,A -85,B 0,C 180,E1 -21897.604,E2 -21897.604} C_VEL
LIN {X 0,Y 203.962,Z 736.96,A -85,B 0,C 180,E1 -21900.219,E2 -21900.219} C_VEL
LIN {X 0,Y 207.479,Z 727.407,A -85,B 0,C 180,E1 -21902.817,E2 -21902.817} C_VEL
LIN {X 0,Y 211.019,Z 716.701,A -85,B 0,C 180,E1 -21905.064,E2 -21905.064} C_VEL
LIN {X 0,Y 214.125,Z 706.026,A -85,B 0,C 180,E1 -21906.797,E2 -21906.797} C_VEL
LIN {X 0,Y 216.898,Z 694.072,A -85,B 0,C 180,E1 -21908.288,E2 -21908.288} C_VEL
LIN {X 0,Y 218.858,Z 683.065,A -85,B 0,C 180,E1 -21909.333,E2 -21909.333} C_VEL
LIN {X 0,Y 220.623,Z 669.727,A -85,B 0,C 180,E1 -21910.219,E2 -21910.219} C_VEL
LIN {X 0,Y 221.693,Z 656.436,A -85,B 0,C 180,E1 -21910.737,E2 -21910.737} C_VEL
LIN {X 0,Y 223.757,Z 614.562,A -85,B 0,C 180,E1 -21912.014,E2 -21912.014} C_VEL
LIN {X 0,Y 216.698,Z 598.691,A -85,B 0,C 180,E1 -21914.294,E2 -21914.294} C_VEL
LIN {X 0,Y 209.884,Z 585.904,A -85,B 0,C 180,E1 -21916.611,E2 -21916.611} C_VEL
LIN {X 0,Y 202.151,Z 574.427,A -85,B 0,C 180,E1 -21919.408,E2 -21919.408} C_VEL
LIN {X 0,Y 199.627,Z 570.741,A -85,B 0,C 180,E1 -21920.399,E2 -21920.399} C_VEL
LIN {X 0,Y 196.824,Z 567.302,A -85,B 0,C 180,E1 -21921.518,E2 -21921.518} C_VEL
LIN {X 0,Y 195.827,Z 565.584,A -85,B 0,C 180,E1 -21921.958,E2 -21921.958} C_VEL
LIN {X 0,Y 193.726,Z 563.552,A -85,B 0,C 180,E1 -21922.822,E2 -21922.822} C_VEL
LIN {X 0,Y 192.702,Z 561.165,A -85,B 0,C 180,E1 -21923.337,E2 -21923.337} C_VEL
LIN {X 0,Y 192.586,Z 560.491,A -85,B 0,C 180,E1 -21923.472,E2 -21923.472} C_VEL
LIN {X 0,Y 192.606,Z 560.489,A -85,B 0,C 180,E1 -21927.059,E2 -21927.059} C_VEL
LIN {X 0,Y 192.662,Z 560.487,A -85,B 0,C 180,E1 -21931.691,E2 -21931.691} C_VEL
LIN {X 0,Y 192.703,Z 560.477,A -85,B 0,C 180,E1 -21936.348,E2 -21936.348} C_VEL
LIN {X 0,Y 192.729,Z 560.469,A -85,B 0,C 180,E1 -21941.457,E2 -21941.457} C_VEL
LIN {X 0,Y 192.76,Z 560.473,A -85,B 0,C 180,E1 -21945.213,E2 -21945.213} C_VEL
LIN {X 0,Y 192.942,Z 560.452,A -85,B 0,C 180,E1 -21949.566,E2 -21949.566} C_VEL
LIN {X 0,Y 192.981,Z 560.438,A -85,B 0,C 180,E1 -21953.727,E2 -21953.727} C_VEL
LIN {X 0,Y 193.259,Z 560.396,A -85,B 0,C 180,E1 -21957.916,E2 -21957.916} C_VEL
LIN {X 0,Y 193.442,Z 560.388,A -85,B 0,C 180,E1 -21960,E2 -21960} C_VEL
LIN {X 0,Y 192.968,Z 560.436,A -85,B 0,C 180,E1 -21964.177,E2 -21964.177} C_VEL
LIN {X 0,Y 193.032,Z 560.426,A -85,B 0,C 180,E1 -21968.374,E2 -21968.374} C_VEL
LIN {X 0,Y 192.8,Z 560.459,A -85,B 0,C 180,E1 -21972.633,E2 -21972.633} C_VEL
LIN {X 0,Y 192.753,Z 560.471,A -85,B 0,C 180,E1 -21976.959,E2 -21976.959} C_VEL
LIN {X 0,Y 192.618,Z 560.49,A -85,B 0,C 180,E1 -21981.399,E2 -21981.399} C_VEL
LIN {X 0,Y 192.644,Z 560.482,A -85,B 0,C 180,E1 -21984.213,E2 -21984.213} C_VEL
LIN {X 0,Y 192.647,Z 560.485,A -85,B 0,C 180,E1 -21988.892,E2 -21988.892} C_VEL
LIN {X 0,Y 192.597,Z 560.495,A -85,B 0,C 180,E1 -21993.186,E2 -21993.186} C_VEL
LIN {X 0,Y 192.593,Z 560.546,A -85,B 0,C 180,E1 -21997.501,E2 -21997.501} C_VEL
LIN {X 0,Y 193.921,Z 564.976,A -85,B 0,C 180,E1 -22000.976,E2 -22000.976} C_VEL
LIN {X 0,Y 196.36,Z 569.05,A -85,B 0,C 180,E1 -22002.065,E2 -22002.065} C_VEL
LIN {X 0,Y 197.885,Z 571.204,A -85,B 0,C 180,E1 -22002.699,E2 -22002.699} C_VEL
LIN {X 0,Y 201.963,Z 577.914,A -85,B 0,C 180,E1 -22004.359,E2 -22004.359} C_VEL
LIN {X 0,Y 206.652,Z 585.688,A -85,B 0,C 180,E1 -22006.131,E2 -22006.131} C_VEL
LIN {X 0,Y 213.249,Z 598.233,A -85,B 0,C 180,E1 -22008.481,E2 -22008.481} C_VEL
LIN {X 0,Y 220.353,Z 614.105,A -85,B 0,C 180,E1 -22010.865,E2 -22010.865} C_VEL
LIN {X 0,Y 222.331,Z 619.194,A -85,B 0,C 180,E1 -22011.514,E2 -22011.514} C_VEL
LIN {X 0,Y 222.442,Z 620.163,A -85,B 0,C 180,E1 -22011.579,E2 -22011.579} C_VEL
LIN {X 0,Y 222.244,Z 624.048,A -85,B 0,C 180,E1 -22011.696,E2 -22011.696} C_VEL
LIN {X 0,Y 220.22,Z 630.38,A -85,B 0,C 180,E1 -22011.519,E2 -22011.519} C_VEL
LIN {X 0,Y 217.843,Z 636.757,A -85,B 0,C 180,E1 -22011.26,E2 -22011.26} C_VEL
LIN {X 0,Y 217.131,Z 640.755,A -85,B 0,C 180,E1 -22011.271,E2 -22011.271} C_VEL
LIN {X 0,Y 215.117,Z 674.654,A -85,B 0,C 180,E1 -22012.339,E2 -22012.339} C_VEL
LIN {X 0,Y 213.369,Z 688.547,A -85,B 0,C 180,E1 -22013.108,E2 -22013.108} C_VEL
LIN {X 0,Y 210.967,Z 701.421,A -85,B 0,C 180,E1 -22014.193,E2 -22014.193} C_VEL
LIN {X 0,Y 208.052,Z 713.093,A -85,B 0,C 180,E1 -22015.542,E2 -22015.542} C_VEL
LIN {X 0,Y 204.817,Z 724.362,A -85,B 0,C 180,E1 -22017.287,E2 -22017.287} C_VEL
LIN {X 0,Y 201.286,Z 734.532,A -85,B 0,C 180,E1 -22019.294,E2 -22019.294} C_VEL
LIN {X 0,Y 197.415,Z 744.5,A -85,B 0,C 180,E1 -22021.856,E2 -22021.856} C_VEL
LIN {X 0,Y 193.776,Z 753.26,A -85,B 0,C 180,E1 -22024.764,E2 -22024.764} C_VEL
LIN {X 0,Y 190.761,Z 760.338,A -85,B 0,C 180,E1 -22027.814,E2 -22027.814} C_VEL
LIN {X 0,Y 187.737,Z 766.79,A -85,B 0,C 180,E1 -22031.446,E2 -22031.446} C_VEL
LIN {X 0,Y 185.706,Z 771.058,A -85,B 0,C 180,E1 -22034.639,E2 -22034.639} C_VEL
LIN {X 0,Y 184.798,Z 773.33,A -85,B 0,C 180,E1 -22036.81,E2 -22036.81} C_VEL
LIN {X 0,Y 184.059,Z 775.149,A -85,B 0,C 180,E1 -22038.994,E2 -22038.994} C_VEL
LIN {X 0,Y 183.212,Z 777.511,A -85,B 0,C 180,E1 -22043.392,E2 -22043.392} C_VEL
LIN {X 0,Y 183.017,Z 778.244,A -85,B 0,C 180,E1 -22046.782,E2 -22046.782} C_VEL
LIN {X 0,Y 183.187,Z 778.074,A -85,B 0,C 180,E1 -22050,E2 -22050} C_VEL
LIN {X 0,Y 183.074,Z 776.882,A -85,B 0,C 180,E1 -22053.523,E2 -22053.523} C_VEL
LIN {X 0,Y 183.211,Z 774.991,A -85,B 0,C 180,E1 -22056.608,E2 -22056.608} C_VEL
LIN {X 0,Y 183.715,Z 772.003,A -85,B 0,C 180,E1 -22059.912,E2 -22059.912} C_VEL
LIN {X 0,Y 184.621,Z 767.958,A -85,B 0,C 180,E1 -22063.203,E2 -22063.203} C_VEL
LIN {X 0,Y 186.417,Z 761.737,A -85,B 0,C 180,E1 -22066.988,E2 -22066.988} C_VEL
